LIN {X 0,Y 307.304,Z 950.743,A -85,B 0,C 180,E1 6847.604,E2 6847.604} C_VEL
LIN {X 0,Y 314.921,Z 929.321,A -85,B 0,C 180,E1 6846.872,E2 6846.872} C_VEL
LIN {X 0,Y 321.32,Z 907.161,A -85,B 0,C 180,E1 6846.28,E2 6846.28} C_VEL
LIN {X 0,Y 326.078,Z 884.655,A -85,B 0,C 180,E1 6845.831,E2 6845.831} C_VEL
LIN {X 0,Y 330.037,Z 856.626,A -85,B 0,C 180,E1 6845.371,E2 6845.371} C_VEL
LIN {X 0,Y 339.234,Z 777.222,A -85,B 0,C 180,E1 6844.099,E2 6844.099} C_VEL
LIN {X 0,Y 338.826,Z 774.8,A -85,B 0,C 180,E1 6841.353,E2 6841.353} C_VEL
LIN {X 0,Y 338.86,Z 775.076,A -85,B 0,C 180,E1 6838.648,E2 6838.648} C_VEL
LIN {X 0,Y 339.251,Z 777.523,A -85,B 0,C 180,E1 6836.249,E2 6836.249} C_VEL
LIN {X 0,Y 331.698,Z 842.7,A -85,B 0,C 180,E1 6835.221,E2 6835.221} C_VEL
LIN {X 0,Y 330.732,Z 850.398,A -85,B 0,C 180,E1 6835.274,E2 6835.274} C_VEL
LIN {X 0,Y 327.738,Z 870.97,A -85,B 0,C 180,E1 6836.04,E2 6836.04} C_VEL
LIN {X 0,Y 326.755,Z 877.56,A -85,B 0,C 180,E1 6836.062,E2 6836.062} C_VEL
LIN {X 0,Y 322.13,Z 901.741,A -85,B 0,C 180,E1 6835.656,E2 6835.656} C_VEL
LIN {X 0,Y 316.056,Z 924.847,A -85,B 0,C 180,E1 6835.216,E2 6835.216} C_VEL
LIN {X 0,Y 308.577,Z 946.561,A -85,B 0,C 180,E1 6834.679,E2 6834.679} C_VEL
LIN {X 0,Y 299.618,Z 968.19,A -85,B 0,C 180,E1 6833.966,E2 6833.966} C_VEL
LIN {X 0,Y 289.561,Z 988.431,A -85,B 0,C 180,E1 6833.093,E2 6833.093} C_VEL
LIN {X 0,Y 277.319,Z 1009.585,A -85,B 0,C 180,E1 6831.917,E2 6831.917} C_VEL
LIN {X 0,Y 265.491,Z 1027.358,A -85,B 0,C 180,E1 6830.648,E2 6830.648} C_VEL
LIN {X 0,Y 251.154,Z 1046.271,A -85,B 0,C 180,E1 6828.911,E2 6828.911} C_VEL
LIN {X 0,Y 237.094,Z 1062.776,A -85,B 0,C 180,E1 6826.946,E2 6826.946} C_VEL
LIN {X 0,Y 222.042,Z 1078.451,A -85,B 0,C 180,E1 6824.503,E2 6824.503} C_VEL
LIN {X 0,Y 206.628,Z 1093.042,A -85,B 0,C 180,E1 6821.519,E2 6821.519} C_VEL
LIN {X 0,Y 190.265,Z 1106.858,A -85,B 0,C 180,E1 6817.652,E2 6817.652} C_VEL
LIN {X 0,Y 174.199,Z 1119.33,A -85,B 0,C 180,E1 6812.83,E2 6812.83} C_VEL
LIN {X 0,Y 160.204,Z 1129.348,A -85,B 0,C 180,E1 6807.41,E2 6807.41} C_VEL
LIN {X 0,Y 145.976,Z 1139.015,A -85,B 0,C 180,E1 6799.922,E2 6799.922} C_VEL
LIN {X 0,Y 135.005,Z 1146.412,A -85,B 0,C 180,E1 6791.583,E2 6791.583} C_VEL
LIN {X 0,Y 126.79,Z 1152.12,A -85,B 0,C 180,E1 6781.894,E2 6781.894} C_VEL
LIN {X 0,Y 122.009,Z 1156.198,A -85,B 0,C 180,E1 6771.639,E2 6771.639} C_VEL
LIN {X 0,Y 120.185,Z 1158.49,A -85,B 0,C 180,E1 6761.516,E2 6761.516} C_VEL
LIN {X 0,Y 120.048,Z 1159.311,A -85,B 0,C 180,E1 6754.298,E2 6754.298} C_VEL
LIN {X 0,Y 120.076,Z 1159.432,A -85,B 0,C 180,E1 6748.09,E2 6748.09} C_VEL
LIN {X 0,Y 120.087,Z 1158.85,A -85,B 0,C 180,E1 6740.897,E2 6740.897} C_VEL
LIN {X 0,Y 121.02,Z 1157.169,A -85,B 0,C 180,E1 6732.199,E2 6732.199} C_VEL
LIN {X 0,Y 124.458,Z 1153.974,A -85,B 0,C 180,E1 6722.227,E2 6722.227} C_VEL
LIN {X 0,Y 131.118,Z 1148.973,A -85,B 0,C 180,E1 6712.405,E2 6712.405} C_VEL
LIN {X 0,Y 141.005,Z 1142.346,A -85,B 0,C 180,E1 6703.456,E2 6703.456} C_VEL
LIN {X 0,Y 153.181,Z 1134.092,A -85,B 0,C 180,E1 6695.962,E2 6695.962} C_VEL
LIN {X 0,Y 167.02,Z 1124.515,A -85,B 0,C 180,E1 6689.767,E2 6689.767} C_VEL
LIN {X 0,Y 182.454,Z 1112.942,A -85,B 0,C 180,E1 6684.535,E2 6684.535} C_VEL
LIN {X 0,Y 199.151,Z 1099.358,A -85,B 0,C 180,E1 6680.137,E2 6680.137} C_VEL
LIN {X 0,Y 214.255,Z 1085.841,A -85,B 0,C 180,E1 6676.925,E2 6676.925} C_VEL
LIN {X 0,Y 229.947,Z 1070.203,A -85,B 0,C 180,E1 6674.148,E2 6674.148} C_VEL
LIN {X 0,Y 244.761,Z 1053.844,A -85,B 0,C 180,E1 6671.935,E2 6671.935} C_VEL
LIN {X 0,Y 258.978,Z 1035.964,A -85,B 0,C 180,E1 6670.096,E2 6670.096} C_VEL
LIN {X 0,Y 272.509,Z 1016.818,A -85,B 0,C 180,E1 6668.57,E2 6668.57} C_VEL
LIN {X 0,Y 284.321,Z 997.516,A -85,B 0,C 180,E1 6667.383,E2 6667.383} C_VEL
LIN {X 0,Y 295.777,Z 975.83,A -85,B 0,C 180,E1 6666.349,E2 6666.349} C_VEL
LIN {X 0,Y 304.435,Z 956.539,A -85,B 0,C 180,E1 6665.639,E2 6665.639} C_VEL
LIN {X 0,Y 312.899,Z 933.827,A -85,B 0,C 180,E1 6664.996,E2 6664.996} C_VEL
LIN {X 0,Y 319.458,Z 911.926,A -85,B 0,C 180,E1 6664.531,E2 6664.531} C_VEL
LIN {X 0,Y 324.641,Z 888.54,A -85,B 0,C 180,E1 6664.12,E2 6664.12} C_VEL
LIN {X 0,Y 328.326,Z 864.356,A -85,B 0,C 180,E1 6663.732,E2 6663.732} C_VEL
LIN {X 0,Y 337.778,Z 783.961,A -85,B 0,C 180,E1 6662.46,E2 6662.46} C_VEL
LIN {X 0,Y 337.616,Z 782.659,A -85,B 0,C 180,E1 6660.848,E2 6660.848} C_VEL
LIN {X 0,Y 337.661,Z 782.798,A -85,B 0,C 180,E1 6658.133,E2 6658.133} C_VEL
LIN {X 0,Y 337.737,Z 784.15,A -85,B 0,C 180,E1 6657.032,E2 6657.032} C_VEL
LIN {X 0,Y 326.505,Z 877.088,A -85,B 0,C 180,E1 6655.607,E2 6655.607} C_VEL
LIN {X 0,Y 321.978,Z 900.285,A -85,B 0,C 180,E1 6655.195,E2 6655.195} C_VEL
LIN {X 0,Y 316.31,Z 921.955,A -85,B 0,C 180,E1 6654.704,E2 6654.704} C_VEL
LIN {X 0,Y 308.915,Z 943.644,A -85,B 0,C 180,E1 6654.055,E2 6654.055} C_VEL
LIN {X 0,Y 300.054,Z 965.186,A -85,B 0,C 180,E1 6653.231,E2 6653.231} C_VEL
LIN {X 0,Y 290.106,Z 985.211,A -85,B 0,C 180,E1 6652.261,E2 6652.261} C_VEL
LIN {X 0,Y 278.377,Z 1005.538,A -85,B 0,C 180,E1 6651.02,E2 6651.02} C_VEL
LIN {X 0,Y 266.782,Z 1022.943,A -85,B 0,C 180,E1 6649.681,E2 6649.681} C_VEL
LIN {X 0,Y 252.163,Z 1042.185,A -85,B 0,C 180,E1 6647.801,E2 6647.801} C_VEL
LIN {X 0,Y 238.725,Z 1057.821,A -85,B 0,C 180,E1 6645.84,E2 6645.84} C_VEL
LIN {X 0,Y 223.427,Z 1073.606,A -85,B 0,C 180,E1 6643.274,E2 6643.274} C_VEL
LIN {X 0,Y 208.212,Z 1087.758,A -85,B 0,C 180,E1 6640.26,E2 6640.26} C_VEL
LIN {X 0,Y 192.835,Z 1100.485,A -85,B 0,C 180,E1 6636.602,E2 6636.602} C_VEL
LIN {X 0,Y 177.611,Z 1112.082,A -85,B 0,C 180,E1 6632.11,E2 6632.11} C_VEL
LIN {X 0,Y 162.914,Z 1122.179,A -85,B 0,C 180,E1 6626.584,E2 6626.584} C_VEL
LIN {X 0,Y 148.74,Z 1131.321,A -85,B 0,C 180,E1 6619.431,E2 6619.431} C_VEL
LIN {X 0,Y 137.683,Z 1138.152,A -85,B 0,C 180,E1 6611.582,E2 6611.582} C_VEL
LIN {X 0,Y 128.647,Z 1143.73,A -85,B 0,C 180,E1 6601.906,E2 6601.906} C_VEL
LIN {X 0,Y 123.388,Z 1147.309,A -85,B 0,C 180,E1 6592.388,E2 6592.388} C_VEL
LIN {X 0,Y 120.712,Z 1149.56,A -85,B 0,C 180,E1 6581.952,E2 6581.952} C_VEL
LIN {X 0,Y 120.131,Z 1150.324,A -85,B 0,C 180,E1 6574.297,E2 6574.297} C_VEL
LIN {X 0,Y 120.103,Z 1150.408,A -85,B 0,C 180,E1 6567.46,E2 6567.46} C_VEL
LIN {X 0,Y 120.536,Z 1149.772,A -85,B 0,C 180,E1 6559.486,E2 6559.486} C_VEL
LIN {X 0,Y 122.361,Z 1148.099,A -85,B 0,C 180,E1 6550.427,E2 6550.427} C_VEL
LIN {X 0,Y 127.569,Z 1144.463,A -85,B 0,C 180,E1 6539.561,E2 6539.561} C_VEL
LIN {X 0,Y 135.249,Z 1139.699,A -85,B 0,C 180,E1 6530.524,E2 6530.524} C_VEL
LIN {X 0,Y 146.433,Z 1132.808,A -85,B 0,C 180,E1 6521.905,E2 6521.905} C_VEL
LIN {X 0,Y 159.565,Z 1124.556,A -85,B 0,C 180,E1 6514.829,E2 6514.829} C_VEL
LIN {X 0,Y 173.885,Z 1114.756,A -85,B 0,C 180,E1 6509.072,E2 6509.072} C_VEL
LIN {X 0,Y 189.62,Z 1103.173,A -85,B 0,C 180,E1 6504.187,E2 6504.187} C_VEL
LIN {X 0,Y 204.821,Z 1090.779,A -85,B 0,C 180,E1 6500.403,E2 6500.403} C_VEL
LIN {X 0,Y 220.887,Z 1076.247,A -85,B 0,C 180,E1 6497.112,E2 6497.112} C_VEL
LIN {X 0,Y 235.551,Z 1061.471,A -85,B 0,C 180,E1 6494.579,E2 6494.579} C_VEL
LIN {X 0,Y 250.283,Z 1044.711,A -85,B 0,C 180,E1 6492.379,E2 6492.379} C_VEL
LIN {X 0,Y 263.957,Z 1027.273,A -85,B 0,C 180,E1 6490.588,E2 6490.588} C_VEL
LIN {X 0,Y 276.451,Z 1008.884,A -85,B 0,C 180,E1 6489.113,E2 6489.113} C_VEL
LIN {X 0,Y 288.167,Z 989.301,A -85,B 0,C 180,E1 6487.861,E2 6487.861} C_VEL
LIN {X 0,Y 298.576,Z 968.744,A -85,B 0,C 180,E1 6486.83,E2 6486.83} C_VEL
LIN {X 0,Y 308.112,Z 946.386,A -85,B 0,C 180,E1 6485.944,E2 6485.944} C_VEL
LIN {X 0,Y 315.308,Z 925.792,A -85,B 0,C 180,E1 6485.31,E2 6485.31} C_VEL
LIN {X 0,Y 321.687,Z 902.515,A -85,B 0,C 180,E1 6484.757,E2 6484.757} C_VEL
LIN {X 0,Y 326.268,Z 880.083,A -85,B 0,C 180,E1 6484.348,E2 6484.348} C_VEL
LIN {X 0,Y 331.506,Z 838.837,A -85,B 0,C 180,E1 6483.708,E2 6483.708} C_VEL
LIN {X 0,Y 337.966,Z 784.117,A -85,B 0,C 180,E1 6482.841,E2 6482.841} C_VEL
LIN {X 0,Y 337.835,Z 782.731,A -85,B 0,C 180,E1 6481.187,E2 6481.187} C_VEL
LIN {X 0,Y 337.865,Z 782.963,A -85,B 0,C 180,E1 6478.813,E2 6478.813} C_VEL
LIN {X 0,Y 337.96,Z 784.492,A -85,B 0,C 180,E1 6477.496,E2 6477.496} C_VEL
LIN {X 0,Y 326.755,Z 877.56,A -85,B 0,C 180,E1 6476.062,E2 6476.062} C_VEL
LIN {X 0,Y 325.501,Z 885.224,A -85,B 0,C 180,E1 6476.117,E2 6476.117} C_VEL
LIN {X 0,Y 321.112,Z 904.429,A -85,B 0,C 180,E1 6476.864,E2 6476.864} C_VEL
LIN {X 0,Y 319.067,Z 911.917,A -85,B 0,C 180,E1 6476.908,E2 6476.908} C_VEL
LIN {X 0,Y 312.544,Z 933.468,A -85,B 0,C 180,E1 6476.483,E2 6476.483} C_VEL
LIN {X 0,Y 304.234,Z 955.616,A -85,B 0,C 180,E1 6475.904,E2 6475.904} C_VEL
LIN {X 0,Y 295.301,Z 975.326,A -85,B 0,C 180,E1 6475.233,E2 6475.233} C_VEL
LIN {X 0,Y 283.871,Z 996.758,A -85,B 0,C 180,E1 6474.284,E2 6474.284} C_VEL
LIN {X 0,Y 272.365,Z 1015.36,A -85,B 0,C 180,E1 6473.223,E2 6473.223} C_VEL
LIN {X 0,Y 258.608,Z 1034.693,A -85,B 0,C 180,E1 6471.798,E2 6471.798} C_VEL
LIN {X 0,Y 244.325,Z 1052.447,A -85,B 0,C 180,E1 6470.104,E2 6470.104} C_VEL
LIN {X 0,Y 228.972,Z 1069.145,A -85,B 0,C 180,E1 6467.999,E2 6467.999} C_VEL
LIN {X 0,Y 212.863,Z 1084.901,A -85,B 0,C 180,E1 6465.379,E2 6465.379} C_VEL
LIN {X 0,Y 197.007,Z 1098.697,A -85,B 0,C 180,E1 6462.272,E2 6462.272} C_VEL
LIN {X 0,Y 179.141,Z 1112.733,A -85,B 0,C 180,E1 6457.896,E2 6457.896} C_VEL
LIN {X 0,Y 163.015,Z 1124.291,A -85,B 0,C 180,E1 6452.792,E2 6452.792} C_VEL
LIN {X 0,Y 148.408,Z 1133.85,A -85,B 0,C 180,E1 6446.658,E2 6446.658} C_VEL
LIN {X 0,Y 135.177,Z 1142.202,A -85,B 0,C 180,E1 6438.977,E2 6438.977} C_VEL
LIN {X 0,Y 124.605,Z 1148.702,A -85,B 0,C 180,E1 6429.936,E2 6429.936} C_VEL
LIN {X 0,Y 116.939,Z 1153.86,A -85,B 0,C 180,E1 6419.166,E2 6419.166} C_VEL
LIN {X 0,Y 113.248,Z 1156.881,A -85,B 0,C 180,E1 6409.066,E2 6409.066} C_VEL
LIN {X 0,Y 112.105,Z 1158.557,A -85,B 0,C 180,E1 6399.755,E2 6399.755} C_VEL
LIN {X 0,Y 112.078,Z 1159.135,A -85,B 0,C 180,E1 6392.044,E2 6392.044} C_VEL
LIN {X 0,Y 112.049,Z 1159.006,A -85,B 0,C 180,E1 6385.392,E2 6385.392} C_VEL
LIN {X 0,Y 112.293,Z 1158.1,A -85,B 0,C 180,E1 6377.137,E2 6377.137} C_VEL
LIN {X 0,Y 114.752,Z 1155.526,A -85,B 0,C 180,E1 6365.824,E2 6365.824} C_VEL
LIN {X 0,Y 120.146,Z 1151.557,A -85,B 0,C 180,E1 6355.534,E2 6355.534} C_VEL
LIN {X 0,Y 129.836,Z 1145.41,A -85,B 0,C 180,E1 6345.11,E2 6345.11} C_VEL
LIN {X 0,Y 141.492,Z 1138.167,A -85,B 0,C 180,E1 6337.009,E2 6337.009} C_VEL
LIN {X 0,Y 156.544,Z 1128.482,A -85,B 0,C 180,E1 6329.696,E2 6329.696} C_VEL
LIN {X 0,Y 172.067,Z 1117.87,A -85,B 0,C 180,E1 6324.171,E2 6324.171} C_VEL
LIN {X 0,Y 188.065,Z 1105.777,A -85,B 0,C 180,E1 6319.771,E2 6319.771} C_VEL
LIN {X 0,Y 204.501,Z 1092.244,A -85,B 0,C 180,E1 6316.181,E2 6316.181} C_VEL
LIN {X 0,Y 219.965,Z 1077.968,A -85,B 0,C 180,E1 6313.403,E2 6313.403} C_VEL
LIN {X 0,Y 236.275,Z 1061.229,A -85,B 0,C 180,E1 6310.954,E2 6310.954} C_VEL
LIN {X 0,Y 249.797,Z 1045.606,A -85,B 0,C 180,E1 6309.213,E2 6309.213} C_VEL
LIN {X 0,Y 264.755,Z 1026.08,A -85,B 0,C 180,E1 6307.538,E2 6307.538} C_VEL
LIN {X 0,Y 276.668,Z 1008.359,A -85,B 0,C 180,E1 6306.361,E2 6306.361} C_VEL
LIN {X 0,Y 288.695,Z 987.722,A -85,B 0,C 180,E1 6305.294,E2 6305.294} C_VEL
LIN {X 0,Y 298.875,Z 967.433,A -85,B 0,C 180,E1 6304.479,E2 6304.479} C_VEL
LIN {X 0,Y 307.649,Z 946.419,A -85,B 0,C 180,E1 6303.833,E2 6303.833} C_VEL
LIN {X 0,Y 315.242,Z 924.604,A -85,B 0,C 180,E1 6303.33,E2 6303.33} C_VEL
LIN {X 0,Y 321.375,Z 901.511,A -85,B 0,C 180,E1 6302.918,E2 6302.918} C_VEL
LIN {X 0,Y 326.058,Z 877.344,A -85,B 0,C 180,E1 6302.531,E2 6302.531} C_VEL
LIN {X 0,Y 336.668,Z 790.79,A -85,B 0,C 180,E1 6301.222,E2 6301.222} C_VEL
LIN {X 0,Y 336.65,Z 790.83,A -85,B 0,C 180,E1 6298.295,E2 6298.295} C_VEL
LIN {X 0,Y 325.954,Z 877.666,A -85,B 0,C 180,E1 6297.005,E2 6297.005} C_VEL
LIN {X 0,Y 321.376,Z 900.726,A -85,B 0,C 180,E1 6296.615,E2 6296.615} C_VEL
LIN {X 0,Y 315.428,Z 923.072,A -85,B 0,C 180,E1 6296.132,E2 6296.132} C_VEL
LIN {X 0,Y 307.903,Z 944.7,A -85,B 0,C 180,E1 6295.516,E2 6295.516} C_VEL
LIN {X 0,Y 298.729,Z 966.492,A -85,B 0,C 180,E1 6294.72,E2 6294.72} C_VEL
LIN {X 0,Y 289.139,Z 985.504,A -85,B 0,C 180,E1 6293.846,E2 6293.846} C_VEL
LIN {X 0,Y 277.23,Z 1005.846,A -85,B 0,C 180,E1 6292.672,E2 6292.672} C_VEL
LIN {X 0,Y 265.592,Z 1023.048,A -85,B 0,C 180,E1 6291.423,E2 6291.423} C_VEL
LIN {X 0,Y 250.946,Z 1042.045,A -85,B 0,C 180,E1 6289.671,E2 6289.671} C_VEL
LIN {X 0,Y 237.31,Z 1057.631,A -85,B 0,C 180,E1 6287.824,E2 6287.824} C_VEL
LIN {X 0,Y 221.205,Z 1073.917,A -85,B 0,C 180,E1 6285.309,E2 6285.309} C_VEL
LIN {X 0,Y 205.579,Z 1088.069,A -85,B 0,C 180,E1 6282.418,E2 6282.418} C_VEL
LIN {X 0,Y 189.711,Z 1100.796,A -85,B 0,C 180,E1 6278.889,E2 6278.889} C_VEL
LIN {X 0,Y 173.459,Z 1112.68,A -85,B 0,C 180,E1 6274.385,E2 6274.385} C_VEL
LIN {X 0,Y 158.507,Z 1122.491,A -85,B 0,C 180,E1 6269.082,E2 6269.082} C_VEL
LIN {X 0,Y 143.497,Z 1131.632,A -85,B 0,C 180,E1 6261.941,E2 6261.941} C_VEL
LIN {X 0,Y 131.914,Z 1138.284,A -85,B 0,C 180,E1 6254.214,E2 6254.214} C_VEL
LIN {X 0,Y 121.749,Z 1144.039,A -85,B 0,C 180,E1 6243.95,E2 6243.95} C_VEL
LIN {X 0,Y 115.679,Z 1147.767,A -85,B 0,C 180,E1 6233.429,E2 6233.429} C_VEL
LIN {X 0,Y 112.813,Z 1149.864,A -85,B 0,C 180,E1 6222.803,E2 6222.803} C_VEL
LIN {X 0,Y 112.147,Z 1150.624,A -85,B 0,C 180,E1 6214.604,E2 6214.604} C_VEL
LIN {X 0,Y 112.108,Z 1150.709,A -85,B 0,C 180,E1 6207.322,E2 6207.322} C_VEL
LIN {X 0,Y 112.559,Z 1150.137,A -85,B 0,C 180,E1 6199.25,E2 6199.25} C_VEL
LIN {X 0,Y 114.395,Z 1148.616,A -85,B 0,C 180,E1 6190.071,E2 6190.071} C_VEL
LIN {X 0,Y 119.724,Z 1145.292,A -85,B 0,C 180,E1 6178.817,E2 6178.817} C_VEL
LIN {X 0,Y 127.629,Z 1140.739,A -85,B 0,C 180,E1 6169.442,E2 6169.442} C_VEL
LIN {X 0,Y 139.883,Z 1133.801,A -85,B 0,C 180,E1 6160.11,E2 6160.11} C_VEL
LIN {X 0,Y 152.96,Z 1126.055,A -85,B 0,C 180,E1 6153.207,E2 6153.207} C_VEL
LIN {X 0,Y 168.523,Z 1116.07,A -85,B 0,C 180,E1 6147.132,E2 6147.132} C_VEL
LIN {X 0,Y 183.984,Z 1105.302,A -85,B 0,C 180,E1 6142.503,E2 6142.503} C_VEL
LIN {X 0,Y 199.983,Z 1092.808,A -85,B 0,C 180,E1 6138.662,E2 6138.662} C_VEL
LIN {X 0,Y 215.864,Z 1079.167,A -85,B 0,C 180,E1 6135.543,E2 6135.543} C_VEL
LIN {X 0,Y 231.216,Z 1064.217,A -85,B 0,C 180,E1 6132.996,E2 6132.996} C_VEL
LIN {X 0,Y 246.823,Z 1047.208,A -85,B 0,C 180,E1 6130.783,E2 6130.783} C_VEL
LIN {X 0,Y 260.246,Z 1030.584,A -85,B 0,C 180,E1 6129.111,E2 6129.111} C_VEL
LIN {X 0,Y 273.865,Z 1011.368,A -85,B 0,C 180,E1 6127.596,E2 6127.596} C_VEL
LIN {X 0,Y 285.349,Z 992.767,A -85,B 0,C 180,E1 6126.438,E2 6126.438} C_VEL
LIN {X 0,Y 296.282,Z 972.035,A -85,B 0,C 180,E1 6125.42,E2 6125.42} C_VEL
LIN {X 0,Y 305.451,Z 951.658,A -85,B 0,C 180,E1 6124.625,E2 6124.625} C_VEL
LIN {X 0,Y 313.355,Z 930.06,A -85,B 0,C 180,E1 6123.963,E2 6123.963} C_VEL
LIN {X 0,Y 319.874,Z 908.122,A -85,B 0,C 180,E1 6123.436,E2 6123.436} C_VEL
LIN {X 0,Y 324.812,Z 885.385,A -85,B 0,C 180,E1 6123.024,E2 6123.024} C_VEL
LIN {X 0,Y 328.839,Z 857.901,A -85,B 0,C 180,E1 6122.604,E2 6122.604} C_VEL
LIN {X 0,Y 336.875,Z 790.916,A -85,B 0,C 180,E1 6121.574,E2 6121.574} C_VEL
LIN {X 0,Y 336.873,Z 790.849,A -85,B 0,C 180,E1 6118.98,E2 6118.98} C_VEL
LIN {X 0,Y 336.844,Z 791.345,A -85,B 0,C 180,E1 6118.754,E2 6118.754} C_VEL
LIN {X 0,Y 326.089,Z 878.773,A -85,B 0,C 180,E1 6117.45,E2 6117.45} C_VEL
LIN {X 0,Y 321.406,Z 902.367,A -85,B 0,C 180,E1 6117.071,E2 6117.071} C_VEL
LIN {X 0,Y 319.067,Z 911.917,A -85,B 0,C 180,E1 6116.908,E2 6116.908} C_VEL
LIN {X 0,Y 316.904,Z 919.36,A -85,B 0,C 180,E1 6116.972,E2 6116.972} C_VEL
LIN {X 0,Y 310.573,Z 938.034,A -85,B 0,C 180,E1 6117.714,E2 6117.714} C_VEL
LIN {X 0,Y 307.761,Z 945.289,A -85,B 0,C 180,E1 6117.695,E2 6117.695} C_VEL
LIN {X 0,Y 298.842,Z 966.585,A -85,B 0,C 180,E1 6117.094,E2 6117.094} C_VEL
LIN {X 0,Y 288.244,Z 987.488,A -85,B 0,C 180,E1 6116.319,E2 6116.319} C_VEL
LIN {X 0,Y 275.883,Z 1008.394,A -85,B 0,C 180,E1 6115.314,E2 6115.314} C_VEL
LIN {X 0,Y 263.804,Z 1026.077,A -85,B 0,C 180,E1 6114.218,E2 6114.218} C_VEL
LIN {X 0,Y 248.986,Z 1045.099,A -85,B 0,C 180,E1 6112.694,E2 6112.694} C_VEL
LIN {X 0,Y 234.845,Z 1061.136,A -85,B 0,C 180,E1 6111.02,E2 6111.02} C_VEL
LIN {X 0,Y 219.105,Z 1076.976,A -85,B 0,C 180,E1 6108.849,E2 6108.849} C_VEL
LIN {X 0,Y 203.74,Z 1090.856,A -85,B 0,C 180,E1 6106.332,E2 6106.332} C_VEL
LIN {X 0,Y 186.261,Z 1104.94,A -85,B 0,C 180,E1 6102.845,E2 6102.845} C_VEL
LIN {X 0,Y 169.034,Z 1117.502,A -85,B 0,C 180,E1 6098.486,E2 6098.486} C_VEL
LIN {X 0,Y 152.563,Z 1128.251,A -85,B 0,C 180,E1 6093.037,E2 6093.037} C_VEL
LIN {X 0,Y 136.211,Z 1138.143,A -85,B 0,C 180,E1 6085.584,E2 6085.584} C_VEL
LIN {X 0,Y 123.71,Z 1145.352,A -85,B 0,C 180,E1 6077.347,E2 6077.347} C_VEL
LIN {X 0,Y 113.387,Z 1151.28,A -85,B 0,C 180,E1 6066.842,E2 6066.842} C_VEL
LIN {X 0,Y 107.073,Z 1155.414,A -85,B 0,C 180,E1 6055.438,E2 6055.438} C_VEL
LIN {X 0,Y 104.383,Z 1157.807,A -85,B 0,C 180,E1 6043.854,E2 6043.854} C_VEL
LIN {X 0,Y 104.046,Z 1158.683,A -85,B 0,C 180,E1 6035.513,E2 6035.513} C_VEL
LIN {X 0,Y 104.088,Z 1158.856,A -85,B 0,C 180,E1 6028.347,E2 6028.347} C_VEL
LIN {X 0,Y 104.112,Z 1158.316,A -85,B 0,C 180,E1 6020.044,E2 6020.044} C_VEL
LIN {X 0,Y 105.448,Z 1156.632,A -85,B 0,C 180,E1 6009.833,E2 6009.833} C_VEL
LIN {X 0,Y 109.782,Z 1153.522,A -85,B 0,C 180,E1 5998.724,E2 5998.724} C_VEL
LIN {X 0,Y 118.321,Z 1148.345,A -85,B 0,C 180,E1 5987.464,E2 5987.464} C_VEL
LIN {X 0,Y 129.828,Z 1141.832,A -85,B 0,C 180,E1 5978.227,E2 5978.227} C_VEL
LIN {X 0,Y 144.319,Z 1133.244,A -85,B 0,C 180,E1 5970.38,E2 5970.38} C_VEL
LIN {X 0,Y 160.125,Z 1123.355,A -85,B 0,C 180,E1 5964.262,E2 5964.262} C_VEL
LIN {X 0,Y 176.208,Z 1112.275,A -85,B 0,C 180,E1 5959.559,E2 5959.559} C_VEL
LIN {X 0,Y 194.03,Z 1098.727,A -85,B 0,C 180,E1 5955.496,E2 5955.496} C_VEL
LIN {X 0,Y 210.01,Z 1085.211,A -85,B 0,C 180,E1 5952.573,E2 5952.573} C_VEL
LIN {X 0,Y 226.466,Z 1069.576,A -85,B 0,C 180,E1 5950.078,E2 5950.078} C_VEL
LIN {X 0,Y 242.218,Z 1052.856,A -85,B 0,C 180,E1 5948.067,E2 5948.067} C_VEL
LIN {X 0,Y 256.607,Z 1035.34,A -85,B 0,C 180,E1 5946.48,E2 5946.48} C_VEL
LIN {X 0,Y 270.554,Z 1016.195,A -85,B 0,C 180,E1 5945.14,E2 5945.14} C_VEL
LIN {X 0,Y 282.689,Z 996.894,A -85,B 0,C 180,E1 5944.103,E2 5944.103} C_VEL
LIN {X 0,Y 294.423,Z 975.209,A -85,B 0,C 180,E1 5943.206,E2 5943.206} C_VEL
LIN {X 0,Y 303.272,Z 955.918,A -85,B 0,C 180,E1 5942.595,E2 5942.595} C_VEL
LIN {X 0,Y 311.909,Z 933.204,A -85,B 0,C 180,E1 5942.044,E2 5942.044} C_VEL
LIN {X 0,Y 318.529,Z 911.517,A -85,B 0,C 180,E1 5941.647,E2 5941.647} C_VEL
LIN {X 0,Y 323.852,Z 888.067,A -85,B 0,C 180,E1 5941.281,E2 5941.281} C_VEL
LIN {X 0,Y 327.641,Z 863.956,A -85,B 0,C 180,E1 5940.925,E2 5940.925} C_VEL
LIN {X 0,Y 335.605,Z 798.522,A -85,B 0,C 180,E1 5939.957,E2 5939.957} C_VEL
LIN {X 0,Y 335.581,Z 798.71,A -85,B 0,C 180,E1 5939.549,E2 5939.549} C_VEL
LIN {X 0,Y 325.6,Z 878.223,A -85,B 0,C 180,E1 5938.407,E2 5938.407} C_VEL
LIN {X 0,Y 320.973,Z 901.168,A -85,B 0,C 180,E1 5938.039,E2 5938.039} C_VEL
LIN {X 0,Y 314.989,Z 923.383,A -85,B 0,C 180,E1 5937.588,E2 5937.588} C_VEL
LIN {X 0,Y 307.38,Z 945.01,A -85,B 0,C 180,E1 5937.008,E2 5937.008} C_VEL
LIN {X 0,Y 298.097,Z 966.801,A -85,B 0,C 180,E1 5936.261,E2 5936.261} C_VEL
LIN {X 0,Y 288.199,Z 986.156,A -85,B 0,C 180,E1 5935.423,E2 5935.423} C_VEL
LIN {X 0,Y 275.833,Z 1006.882,A -85,B 0,C 180,E1 5934.291,E2 5934.291} C_VEL
LIN {X 0,Y 263.88,Z 1024.221,A -85,B 0,C 180,E1 5933.096,E2 5933.096} C_VEL
LIN {X 0,Y 249.195,Z 1042.842,A -85,B 0,C 180,E1 5931.462,E2 5931.462} C_VEL
LIN {X 0,Y 235.399,Z 1058.289,A -85,B 0,C 180,E1 5929.723,E2 5929.723} C_VEL
LIN {X 0,Y 219.269,Z 1074.227,A -85,B 0,C 180,E1 5927.383,E2 5927.383} C_VEL
LIN {X 0,Y 202.936,Z 1088.649,A -85,B 0,C 180,E1 5924.57,E2 5924.57} C_VEL
LIN {X 0,Y 186.057,Z 1101.73,A -85,B 0,C 180,E1 5921.055,E2 5921.055} C_VEL
LIN {X 0,Y 168.913,Z 1113.711,A -85,B 0,C 180,E1 5916.566,E2 5916.566} C_VEL
LIN {X 0,Y 153.688,Z 1123.25,A -85,B 0,C 180,E1 5911.438,E2 5911.438} C_VEL
LIN {X 0,Y 137.907,Z 1132.286,A -85,B 0,C 180,E1 5904.296,E2 5904.296} C_VEL
LIN {X 0,Y 125.067,Z 1139.18,A -85,B 0,C 180,E1 5896.016,E2 5896.016} C_VEL
LIN {X 0,Y 114.637,Z 1144.545,A -85,B 0,C 180,E1 5885.76,E2 5885.76} C_VEL
LIN {X 0,Y 108.013,Z 1148.225,A -85,B 0,C 180,E1 5874.619,E2 5874.619} C_VEL
LIN {X 0,Y 104.861,Z 1150.229,A -85,B 0,C 180,E1 5863.23,E2 5863.23} C_VEL
LIN {X 0,Y 104.144,Z 1150.945,A -85,B 0,C 180,E1 5854.406,E2 5854.406} C_VEL
LIN {X 0,Y 104.115,Z 1151.011,A -85,B 0,C 180,E1 5847.159,E2 5847.159} C_VEL
LIN {X 0,Y 104.645,Z 1150.439,A -85,B 0,C 180,E1 5838.426,E2 5838.426} C_VEL
LIN {X 0,Y 106.777,Z 1148.921,A -85,B 0,C 180,E1 5828.581,E2 5828.581} C_VEL
LIN {X 0,Y 112.78,Z 1145.599,A -85,B 0,C 180,E1 5816.657,E2 5816.657} C_VEL
LIN {X 0,Y 121.478,Z 1141.048,A -85,B 0,C 180,E1 5806.911,E2 5806.911} C_VEL
LIN {X 0,Y 134.699,Z 1134.11,A -85,B 0,C 180,E1 5797.416,E2 5797.416} C_VEL
LIN {X 0,Y 148.587,Z 1126.364,A -85,B 0,C 180,E1 5790.535,E2 5790.535} C_VEL
LIN {X 0,Y 164.915,Z 1116.379,A -85,B 0,C 180,E1 5784.574,E2 5784.574} C_VEL
LIN {X 0,Y 181.397,Z 1105.327,A -85,B 0,C 180,E1 5779.984,E2 5779.984} C_VEL
LIN {X 0,Y 197.938,Z 1092.768,A -85,B 0,C 180,E1 5776.31,E2 5776.31} C_VEL
LIN {X 0,Y 214.705,Z 1078.639,A -85,B 0,C 180,E1 5773.273,E2 5773.273} C_VEL
LIN {X 0,Y 230.133,Z 1063.906,A -85,B 0,C 180,E1 5770.918,E2 5770.918} C_VEL
LIN {X 0,Y 246.364,Z 1046.413,A -85,B 0,C 180,E1 5768.799,E2 5768.799} C_VEL
LIN {X 0,Y 260.033,Z 1029.681,A -85,B 0,C 180,E1 5767.234,E2 5767.234} C_VEL
LIN {X 0,Y 273.391,Z 1010.938,A -85,B 0,C 180,E1 5765.864,E2 5765.864} C_VEL
LIN {X 0,Y 285.277,Z 991.866,A -85,B 0,C 180,E1 5764.759,E2 5764.759} C_VEL
LIN {X 0,Y 295.973,Z 971.628,A -85,B 0,C 180,E1 5763.836,E2 5763.836} C_VEL
LIN {X 0,Y 305.398,Z 950.797,A -85,B 0,C 180,E1 5763.08,E2 5763.08} C_VEL
LIN {X 0,Y 313.247,Z 929.321,A -85,B 0,C 180,E1 5762.471,E2 5762.471} C_VEL
LIN {X 0,Y 319.819,Z 907.043,A -85,B 0,C 180,E1 5761.977,E2 5761.977} C_VEL
LIN {X 0,Y 324.609,Z 885.036,A -85,B 0,C 180,E1 5761.603,E2 5761.603} C_VEL
LIN {X 0,Y 329.038,Z 854.344,A -85,B 0,C 180,E1 5761.155,E2 5761.155} C_VEL
LIN {X 0,Y 335.84,Z 798.602,A -85,B 0,C 180,E1 5760.342,E2 5760.342} C_VEL
LIN {X 0,Y 335.817,Z 798.811,A -85,B 0,C 180,E1 5760.012,E2 5760.012} C_VEL
LIN {X 0,Y 325.8,Z 878.707,A -85,B 0,C 180,E1 5758.86,E2 5758.86} C_VEL
LIN {X 0,Y 321.064,Z 902.209,A -85,B 0,C 180,E1 5758.503,E2 5758.503} C_VEL
LIN {X 0,Y 314.874,Z 925.007,A -85,B 0,C 180,E1 5758.123,E2 5758.123} C_VEL
LIN {X 0,Y 307.761,Z 945.289,A -85,B 0,C 180,E1 5757.695,E2 5757.695} C_VEL
LIN {X 0,Y 304.859,Z 952.654,A -85,B 0,C 180,E1 5757.699,E2 5757.699} C_VEL
LIN {X 0,Y 296.472,Z 970.607,A -85,B 0,C 180,E1 5758.327,E2 5758.327} C_VEL
LIN {X 0,Y 293.07,Z 977.439,A -85,B 0,C 180,E1 5758.292,E2 5758.292} C_VEL
LIN {X 0,Y 281.728,Z 997.792,A -85,B 0,C 180,E1 5757.499,E2 5757.499} C_VEL
LIN {X 0,Y 269.454,Z 1016.979,A -85,B 0,C 180,E1 5756.537,E2 5756.537} C_VEL
LIN {X 0,Y 255.81,Z 1035.313,A -85,B 0,C 180,E1 5755.337,E2 5755.337} C_VEL
LIN {X 0,Y 241.342,Z 1052.622,A -85,B 0,C 180,E1 5753.878,E2 5753.878} C_VEL
LIN {X 0,Y 226.109,Z 1068.53,A -85,B 0,C 180,E1 5752.107,E2 5752.107} C_VEL
LIN {X 0,Y 209.284,Z 1084.282,A -85,B 0,C 180,E1 5749.79,E2 5749.79} C_VEL
LIN {X 0,Y 192.867,Z 1097.846,A -85,B 0,C 180,E1 5747.064,E2 5747.064} C_VEL
LIN {X 0,Y 174.389,Z 1111.522,A -85,B 0,C 180,E1 5743.233,E2 5743.233} C_VEL
LIN {X 0,Y 157.674,Z 1122.61,A -85,B 0,C 180,E1 5738.774,E2 5738.774} C_VEL
LIN {X 0,Y 140.612,Z 1132.805,A -85,B 0,C 180,E1 5732.727,E2 5732.727} C_VEL
LIN {X 0,Y 125.45,Z 1141.252,A -85,B 0,C 180,E1 5725.177,E2 5725.177} C_VEL
LIN {X 0,Y 112.812,Z 1147.812,A -85,B 0,C 180,E1 5715.881,E2 5715.881} C_VEL
LIN {X 0,Y 103.105,Z 1153.069,A -85,B 0,C 180,E1 5704.225,E2 5704.225} C_VEL
LIN {X 0,Y 97.893,Z 1156.266,A -85,B 0,C 180,E1 5692.203,E2 5692.203} C_VEL
LIN {X 0,Y 96.143,Z 1158.024,A -85,B 0,C 180,E1 5680.788,E2 5680.788} C_VEL
LIN {X 0,Y 96.09,Z 1158.56,A -85,B 0,C 180,E1 5671.788,E2 5671.788} C_VEL
LIN {X 0,Y 96.051,Z 1158.378,A -85,B 0,C 180,E1 5664.024,E2 5664.024} C_VEL
LIN {X 0,Y 96.652,Z 1157.338,A -85,B 0,C 180,E1 5653.779,E2 5653.779} C_VEL
LIN {X 0,Y 100.431,Z 1154.568,A -85,B 0,C 180,E1 5640.8,E2 5640.8} C_VEL
LIN {X 0,Y 107.683,Z 1150.497,A -85,B 0,C 180,E1 5629.459,E2 5629.459} C_VEL
LIN {X 0,Y 119.932,Z 1144.037,A -85,B 0,C 180,E1 5618.4,E2 5618.4} C_VEL
LIN {X 0,Y 134.151,Z 1136.439,A -85,B 0,C 180,E1 5610.164,E2 5610.164} C_VEL
LIN {X 0,Y 150.498,Z 1126.906,A -85,B 0,C 180,E1 5603.531,E2 5603.531} C_VEL
LIN {X 0,Y 167.629,Z 1116.066,A -85,B 0,C 180,E1 5598.428,E2 5598.428} C_VEL
LIN {X 0,Y 183.968,Z 1104.498,A -85,B 0,C 180,E1 5594.661,E2 5594.661} C_VEL
LIN {X 0,Y 201.931,Z 1090.379,A -85,B 0,C 180,E1 5591.36,E2 5591.36} C_VEL
LIN {X 0,Y 217.755,Z 1076.385,A -85,B 0,C 180,E1 5588.981,E2 5588.981} C_VEL
LIN {X 0,Y 235.123,Z 1059.063,A -85,B 0,C 180,E1 5586.799,E2 5586.799} C_VEL
LIN {X 0,Y 250.004,Z 1042.293,A -85,B 0,C 180,E1 5585.215,E2 5585.215} C_VEL
LIN {X 0,Y 264.08,Z 1024.109,A -85,B 0,C 180,E1 5583.907,E2 5583.907} C_VEL
LIN {X 0,Y 276.763,Z 1005.59,A -85,B 0,C 180,E1 5582.874,E2 5582.874} C_VEL
LIN {X 0,Y 288.145,Z 986.195,A -85,B 0,C 180,E1 5582.034,E2 5582.034} C_VEL
LIN {X 0,Y 298.56,Z 965.765,A -85,B 0,C 180,E1 5581.343,E2 5581.343} C_VEL
LIN {X 0,Y 307.49,Z 944.507,A -85,B 0,C 180,E1 5580.794,E2 5580.794} C_VEL
LIN {X 0,Y 315.347,Z 921.844,A -85,B 0,C 180,E1 5580.363,E2 5580.363} C_VEL
LIN {X 0,Y 321.268,Z 899.587,A -85,B 0,C 180,E1 5580.027,E2 5580.027} C_VEL
LIN {X 0,Y 324.868,Z 882.043,A -85,B 0,C 180,E1 5579.765,E2 5579.765} C_VEL
LIN {X 0,Y 320.225,Z 903.872,A -85,B 0,C 180,E1 5579.427,E2 5579.427} C_VEL
LIN {X 0,Y 313.512,Z 927.377,A -85,B 0,C 180,E1 5578.959,E2 5578.959} C_VEL
LIN {X 0,Y 306.076,Z 947.874,A -85,B 0,C 180,E1 5578.431,E2 5578.431} C_VEL
LIN {X 0,Y 296.201,Z 970.104,A -85,B 0,C 180,E1 5577.697,E2 5577.697} C_VEL
LIN {X 0,Y 285.398,Z 990.603,A -85,B 0,C 180,E1 5576.839,E2 5576.839} C_VEL
LIN {X 0,Y 273.244,Z 1010.037,A -85,B 0,C 180,E1 5575.803,E2 5575.803} C_VEL
LIN {X 0,Y 260.136,Z 1028.438,A -85,B 0,C 180,E1 5574.566,E2 5574.566} C_VEL
LIN {X 0,Y 246.113,Z 1045.458,A -85,B 0,C 180,E1 5573.102,E2 5573.102} C_VEL
LIN {X 0,Y 230.65,Z 1062.12,A -85,B 0,C 180,E1 5571.259,E2 5571.259} C_VEL
LIN {X 0,Y 214.862,Z 1077.035,A -85,B 0,C 180,E1 5569.083,E2 5569.083} C_VEL
LIN {X 0,Y 196.739,Z 1092.181,A -85,B 0,C 180,E1 5566.098,E2 5566.098} C_VEL
LIN {X 0,Y 180.095,Z 1104.533,A -85,B 0,C 180,E1 5562.733,E2 5562.733} C_VEL
LIN {X 0,Y 162.995,Z 1115.746,A -85,B 0,C 180,E1 5558.403,E2 5558.403} C_VEL
LIN {X 0,Y 146.875,Z 1125.348,A -85,B 0,C 180,E1 5553.101,E2 5553.101} C_VEL
LIN {X 0,Y 131.231,Z 1133.623,A -85,B 0,C 180,E1 5546.151,E2 5546.151} C_VEL
LIN {X 0,Y 117.257,Z 1140.544,A -85,B 0,C 180,E1 5537.168,E2 5537.168} C_VEL
LIN {X 0,Y 107.246,Z 1145.248,A -85,B 0,C 180,E1 5527.303,E2 5527.303} C_VEL
LIN {X 0,Y 99.692,Z 1148.977,A -85,B 0,C 180,E1 5514.282,E2 5514.282} C_VEL
LIN {X 0,Y 96.833,Z 1150.657,A -85,B 0,C 180,E1 5503.132,E2 5503.132} C_VEL
LIN {X 0,Y 96.128,Z 1151.286,A -85,B 0,C 180,E1 5493.579,E2 5493.579} C_VEL
LIN {X 0,Y 96.139,Z 1151.273,A -85,B 0,C 180,E1 5485.826,E2 5485.826} C_VEL
LIN {X 0,Y 96.903,Z 1150.617,A -85,B 0,C 180,E1 5476.273,E2 5476.273} C_VEL
LIN {X 0,Y 100.121,Z 1148.803,A -85,B 0,C 180,E1 5464.57,E2 5464.57} C_VEL
LIN {X 0,Y 107.6,Z 1145.118,A -85,B 0,C 180,E1 5452.173,E2 5452.173} C_VEL
LIN {X 0,Y 118.847,Z 1139.878,A -85,B 0,C 180,E1 5441.518,E2 5441.518} C_VEL
LIN {X 0,Y 132.494,Z 1133.052,A -85,B 0,C 180,E1 5433.108,E2 5433.108} C_VEL
LIN {X 0,Y 148.309,Z 1124.595,A -85,B 0,C 180,E1 5426.28,E2 5426.28} C_VEL
LIN {X 0,Y 164.087,Z 1115.179,A -85,B 0,C 180,E1 5421.205,E2 5421.205} C_VEL
LIN {X 0,Y 182.612,Z 1102.85,A -85,B 0,C 180,E1 5416.63,E2 5416.63} C_VEL
LIN {X 0,Y 199.531,Z 1090.194,A -85,B 0,C 180,E1 5413.328,E2 5413.328} C_VEL
LIN {X 0,Y 215.974,Z 1076.222,A -85,B 0,C 180,E1 5410.672,E2 5410.672} C_VEL
LIN {X 0,Y 231.54,Z 1061.469,A -85,B 0,C 180,E1 5408.55,E2 5408.55} C_VEL
LIN {X 0,Y 246.761,Z 1044.973,A -85,B 0,C 180,E1 5406.749,E2 5406.749} C_VEL
LIN {X 0,Y 261.065,Z 1027.545,A -85,B 0,C 180,E1 5405.266,E2 5405.266} C_VEL
LIN {X 0,Y 274.143,Z 1009.052,A -85,B 0,C 180,E1 5404.042,E2 5404.042} C_VEL
LIN {X 0,Y 286.4,Z 989.212,A -85,B 0,C 180,E1 5403.002,E2 5403.002} C_VEL
LIN {X 0,Y 296.675,Z 969.632,A -85,B 0,C 180,E1 5402.191,E2 5402.191} C_VEL
LIN {X 0,Y 306.76,Z 946.737,A -85,B 0,C 180,E1 5401.442,E2 5401.442} C_VEL
LIN {X 0,Y 314.286,Z 925.809,A -85,B 0,C 180,E1 5400.912,E2 5400.912} C_VEL
LIN {X 0,Y 320.715,Z 902.857,A -85,B 0,C 180,E1 5400.465,E2 5400.465} C_VEL
LIN {X 0,Y 324.507,Z 885.204,A -85,B 0,C 180,E1 5400.18,E2 5400.18} C_VEL
LIN {X 0,Y 319.474,Z 908.115,A -85,B 0,C 180,E1 5399.848,E2 5399.848} C_VEL
LIN {X 0,Y 312.693,Z 930.728,A -85,B 0,C 180,E1 5399.479,E2 5399.479} C_VEL
LIN {X 0,Y 304.502,Z 952.752,A -85,B 0,C 180,E1 5399.013,E2 5399.013} C_VEL
LIN {X 0,Y 295.069,Z 973.359,A -85,B 0,C 180,E1 5398.429,E2 5398.429} C_VEL
LIN {X 0,Y 293.07,Z 977.439,A -85,B 0,C 180,E1 5398.292,E2 5398.292} C_VEL
LIN {X 0,Y 289.494,Z 984.33,A -85,B 0,C 180,E1 5398.243,E2 5398.243} C_VEL
LIN {X 0,Y 279.225,Z 1001.427,A -85,B 0,C 180,E1 5398.783,E2 5398.783} C_VEL
LIN {X 0,Y 274.968,Z 1007.885,A -85,B 0,C 180,E1 5398.701,E2 5398.701} C_VEL
LIN {X 0,Y 262.66,Z 1025.471,A -85,B 0,C 180,E1 5397.78,E2 5397.78} C_VEL
LIN {X 0,Y 247.431,Z 1044.488,A -85,B 0,C 180,E1 5396.481,E2 5396.481} C_VEL
LIN {X 0,Y 232.353,Z 1061.035,A -85,B 0,C 180,E1 5394.993,E2 5394.993} C_VEL
LIN {X 0,Y 215.555,Z 1077.216,A -85,B 0,C 180,E1 5393.046,E2 5393.046} C_VEL
LIN {X 0,Y 198.592,Z 1091.802,A -85,B 0,C 180,E1 5390.682,E2 5390.682} C_VEL
LIN {X 0,Y 181.126,Z 1104.964,A -85,B 0,C 180,E1 5387.708,E2 5387.708} C_VEL
LIN {X 0,Y 163.388,Z 1117.024,A -85,B 0,C 180,E1 5383.896,E2 5383.896} C_VEL
LIN {X 0,Y 145.716,Z 1127.624,A -85,B 0,C 180,E1 5378.936,E2 5378.936} C_VEL
LIN {X 0,Y 127.926,Z 1137.291,A -85,B 0,C 180,E1 5372.029,E2 5372.029} C_VEL
LIN {X 0,Y 113.656,Z 1144.411,A -85,B 0,C 180,E1 5364.031,E2 5364.031} C_VEL
LIN {X 0,Y 100.715,Z 1150.582,A -85,B 0,C 180,E1 5352.725,E2 5352.725} C_VEL
LIN {X 0,Y 92.434,Z 1154.796,A -85,B 0,C 180,E1 5339.839,E2 5339.839} C_VEL
LIN {X 0,Y 88.562,Z 1157.272,A -85,B 0,C 180,E1 5325.72,E2 5325.72} C_VEL
LIN {X 0,Y 88.055,Z 1158.107,A -85,B 0,C 180,E1 5315.864,E2 5315.864} C_VEL
LIN {X 0,Y 88.091,Z 1158.255,A -85,B 0,C 180,E1 5308.047,E2 5308.047} C_VEL
LIN {X 0,Y 88.156,Z 1157.782,A -85,B 0,C 180,E1 5298.881,E2 5298.881} C_VEL
LIN {X 0,Y 90.151,Z 1156.06,A -85,B 0,C 180,E1 5286.466,E2 5286.466} C_VEL
LIN {X 0,Y 95.974,Z 1152.898,A -85,B 0,C 180,E1 5273.569,E2 5273.569} C_VEL
LIN {X 0,Y 106.611,Z 1147.717,A -85,B 0,C 180,E1 5261.383,E2 5261.383} C_VEL
LIN {X 0,Y 120.855,Z 1140.871,A -85,B 0,C 180,E1 5251.552,E2 5251.552} C_VEL
LIN {X 0,Y 137.037,Z 1132.371,A -85,B 0,C 180,E1 5244.115,E2 5244.115} C_VEL
LIN {X 0,Y 154.833,Z 1122.195,A -85,B 0,C 180,E1 5238.324,E2 5238.324} C_VEL
LIN {X 0,Y 172.159,Z 1111.092,A -85,B 0,C 180,E1 5234.09,E2 5234.09} C_VEL
LIN {X 0,Y 191.172,Z 1097.383,A -85,B 0,C 180,E1 5230.491,E2 5230.491} C_VEL
LIN {X 0,Y 208.918,Z 1083.014,A -85,B 0,C 180,E1 5227.821,E2 5227.821} C_VEL
LIN {X 0,Y 225.123,Z 1068.011,A -85,B 0,C 180,E1 5225.797,E2 5225.797} C_VEL
LIN {X 0,Y 241.091,Z 1051.523,A -85,B 0,C 180,E1 5224.113,E2 5224.113} C_VEL
LIN {X 0,Y 255.562,Z 1034.359,A -85,B 0,C 180,E1 5222.791,E2 5222.791} C_VEL
LIN {X 0,Y 270.076,Z 1014.832,A -85,B 0,C 180,E1 5221.64,E2 5221.64} C_VEL
LIN {X 0,Y 281.992,Z 996.273,A -85,B 0,C 180,E1 5220.799,E2 5220.799} C_VEL
LIN {X 0,Y 293.963,Z 974.587,A -85,B 0,C 180,E1 5220.045,E2 5220.045} C_VEL
LIN {X 0,Y 301.34,Z 958.996,A -85,B 0,C 180,E1 5219.619,E2 5219.619} C_VEL
LIN {X 0,Y 291.017,Z 980.191,A -85,B 0,C 180,E1 5218.895,E2 5218.895} C_VEL
LIN {X 0,Y 280.12,Z 999.01,A -85,B 0,C 180,E1 5218.087,E2 5218.087} C_VEL
LIN {X 0,Y 266.34,Z 1019.549,A -85,B 0,C 180,E1 5216.963,E2 5216.963} C_VEL
LIN {X 0,Y 253.157,Z 1036.573,A -85,B 0,C 180,E1 5215.772,E2 5215.772} C_VEL
LIN {X 0,Y 237.206,Z 1054.557,A -85,B 0,C 180,E1 5214.149,E2 5214.149} C_VEL
LIN {X 0,Y 220.996,Z 1070.649,A -85,B 0,C 180,E1 5212.24,E2 5212.24} C_VEL
LIN {X 0,Y 204.132,Z 1085.213,A -85,B 0,C 180,E1 5209.91,E2 5209.91} C_VEL
LIN {X 0,Y 186.703,Z 1098.653,A -85,B 0,C 180,E1 5207.001,E2 5207.001} C_VEL
LIN {X 0,Y 169.061,Z 1110.551,A -85,B 0,C 180,E1 5203.359,E2 5203.359} C_VEL
LIN {X 0,Y 150.531,Z 1121.64,A -85,B 0,C 180,E1 5198.424,E2 5198.424} C_VEL
LIN {X 0,Y 134.091,Z 1130.401,A -85,B 0,C 180,E1 5192.542,E2 5192.542} C_VEL
LIN {X 0,Y 118.645,Z 1137.755,A -85,B 0,C 180,E1 5184.833,E2 5184.833} C_VEL
LIN {X 0,Y 105.17,Z 1143.778,A -85,B 0,C 180,E1 5174.713,E2 5174.713} C_VEL
LIN {X 0,Y 95.289,Z 1147.932,A -85,B 0,C 180,E1 5162.355,E2 5162.355} C_VEL
LIN {X 0,Y 89.878,Z 1150.527,A -85,B 0,C 180,E1 5148.823,E2 5148.823} C_VEL
LIN {X 0,Y 88.261,Z 1151.487,A -85,B 0,C 180,E1 5137.16,E2 5137.16} C_VEL
LIN {X 0,Y 88.119,Z 1151.657,A -85,B 0,C 180,E1 5128.051,E2 5128.051} C_VEL
LIN {X 0,Y 88.715,Z 1151.17,A -85,B 0,C 180,E1 5117.636,E2 5117.636} C_VEL
LIN {X 0,Y 91.56,Z 1149.638,A -85,B 0,C 180,E1 5105.484,E2 5105.484} C_VEL
LIN {X 0,Y 98.628,Z 1146.607,A -85,B 0,C 180,E1 5092.538,E2 5092.538} C_VEL
LIN {X 0,Y 109.432,Z 1141.909,A -85,B 0,C 180,E1 5081.479,E2 5081.479} C_VEL
LIN {X 0,Y 123.944,Z 1135.413,A -85,B 0,C 180,E1 5072.11,E2 5072.11} C_VEL
LIN {X 0,Y 139.342,Z 1127.77,A -85,B 0,C 180,E1 5065.296,E2 5065.296} C_VEL
LIN {X 0,Y 157.909,Z 1117.499,A -85,B 0,C 180,E1 5059.363,E2 5059.363} C_VEL
LIN {X 0,Y 175.112,Z 1106.787,A -85,B 0,C 180,E1 5055.214,E2 5055.214} C_VEL
LIN {X 0,Y 193.045,Z 1094.069,A -85,B 0,C 180,E1 5051.791,E2 5051.791} C_VEL
LIN {X 0,Y 210.606,Z 1080.082,A -85,B 0,C 180,E1 5049.075,E2 5049.075} C_VEL
LIN {X 0,Y 226.649,Z 1065.427,A -85,B 0,C 180,E1 5046.984,E2 5046.984} C_VEL
LIN {X 0,Y 242.953,Z 1048.663,A -85,B 0,C 180,E1 5045.17,E2 5045.17} C_VEL
LIN {X 0,Y 257.002,Z 1032.118,A -85,B 0,C 180,E1 5043.793,E2 5043.793} C_VEL
LIN {X 0,Y 271.442,Z 1012.679,A -85,B 0,C 180,E1 5042.534,E2 5042.534} C_VEL
LIN {X 0,Y 283.071,Z 994.611,A -85,B 0,C 180,E1 5041.611,E2 5041.611} C_VEL
LIN {X 0,Y 294.444,Z 974.003,A -85,B 0,C 180,E1 5040.779,E2 5040.779} C_VEL
LIN {X 0,Y 300.82,Z 960.728,A -85,B 0,C 180,E1 5040.332,E2 5040.332} C_VEL
LIN {X 0,Y 289.963,Z 982.705,A -85,B 0,C 180,E1 5039.696,E2 5039.696} C_VEL
LIN {X 0,Y 278.833,Z 1001.859,A -85,B 0,C 180,E1 5038.973,E2 5038.973} C_VEL
LIN {X 0,Y 274.968,Z 1007.885,A -85,B 0,C 180,E1 5038.701,E2 5038.701} C_VEL
LIN {X 0,Y 270.562,Z 1014.412,A -85,B 0,C 180,E1 5038.6,E2 5038.6} C_VEL
LIN {X 0,Y 258.541,Z 1030.417,A -85,B 0,C 180,E1 5039.053,E2 5039.053} C_VEL
LIN {X 0,Y 253.719,Z 1036.289,A -85,B 0,C 180,E1 5038.918,E2 5038.918} C_VEL
LIN {X 0,Y 237.186,Z 1055.087,A -85,B 0,C 180,E1 5037.532,E2 5037.532} C_VEL
LIN {X 0,Y 221.51,Z 1070.729,A -85,B 0,C 180,E1 5035.991,E2 5035.991} C_VEL
LIN {X 0,Y 204.102,Z 1086.011,A -85,B 0,C 180,E1 5033.963,E2 5033.963} C_VEL
LIN {X 0,Y 187.007,Z 1099.364,A -85,B 0,C 180,E1 5031.542,E2 5031.542} C_VEL
LIN {X 0,Y 168.489,Z 1112.069,A -85,B 0,C 180,E1 5028.278,E2 5028.278} C_VEL
LIN {X 0,Y 149.789,Z 1123.54,A -85,B 0,C 180,E1 5023.988,E2 5023.988} C_VEL
LIN {X 0,Y 132.126,Z 1133.013,A -85,B 0,C 180,E1 5018.558,E2 5018.558} C_VEL
LIN {X 0,Y 114.513,Z 1141.578,A -85,B 0,C 180,E1 5010.824,E2 5010.824} C_VEL
LIN {X 0,Y 100.681,Z 1147.718,A -85,B 0,C 180,E1 5001.677,E2 5001.677} C_VEL
LIN {X 0,Y 88.605,Z 1152.958,A -85,B 0,C 180,E1 4988.362,E2 4988.362} C_VEL
LIN {X 0,Y 82.465,Z 1155.896,A -85,B 0,C 180,E1 4975.109,E2 4975.109} C_VEL
LIN {X 0,Y 80.142,Z 1157.632,A -85,B 0,C 180,E1 4960.784,E2 4960.784} C_VEL
LIN {X 0,Y 80.108,Z 1158.007,A -85,B 0,C 180,E1 4950.714,E2 4950.714} C_VEL
LIN {X 0,Y 80.081,Z 1157.719,A -85,B 0,C 180,E1 4941.381,E2 4941.381} C_VEL
LIN {X 0,Y 81.875,Z 1156.241,A -85,B 0,C 180,E1 4926.995,E2 4926.995} C_VEL
LIN {X 0,Y 87.824,Z 1153.267,A -85,B 0,C 180,E1 4912.884,E2 4912.884} C_VEL
LIN {X 0,Y 98.926,Z 1148.465,A -85,B 0,C 180,E1 4899.81,E2 4899.81} C_VEL
LIN {X 0,Y 113.088,Z 1142.146,A -85,B 0,C 180,E1 4889.947,E2 4889.947} C_VEL
LIN {X 0,Y 131.317,Z 1133.345,A -85,B 0,C 180,E1 4881.73,E2 4881.73} C_VEL
LIN {X 0,Y 148.922,Z 1123.919,A -85,B 0,C 180,E1 4876.235,E2 4876.235} C_VEL
LIN {X 0,Y 167.58,Z 1112.534,A -85,B 0,C 180,E1 4871.898,E2 4871.898} C_VEL
LIN {X 0,Y 186.068,Z 1099.921,A -85,B 0,C 180,E1 4868.597,E2 4868.597} C_VEL
LIN {X 0,Y 203.144,Z 1086.617,A -85,B 0,C 180,E1 4866.15,E2 4866.15} C_VEL
LIN {X 0,Y 220.538,Z 1071.45,A -85,B 0,C 180,E1 4864.104,E2 4864.104} C_VEL
LIN {X 0,Y 236.204,Z 1055.871,A -85,B 0,C 180,E1 4862.546,E2 4862.546} C_VEL
LIN {X 0,Y 253.017,Z 1036.862,A -85,B 0,C 180,E1 4861.126,E2 4861.126} C_VEL
LIN {X 0,Y 266.967,Z 1018.769,A -85,B 0,C 180,E1 4860.107,E2 4860.107} C_VEL
LIN {X 0,Y 276.501,Z 1004.856,A -85,B 0,C 180,E1 4859.485,E2 4859.485} C_VEL
LIN {X 0,Y 263.555,Z 1023.165,A -85,B 0,C 180,E1 4858.512,E2 4858.512} C_VEL
LIN {X 0,Y 249.244,Z 1040.987,A -85,B 0,C 180,E1 4857.307,E2 4857.307} C_VEL
LIN {X 0,Y 234.565,Z 1056.869,A -85,B 0,C 180,E1 4855.921,E2 4855.921} C_VEL
LIN {X 0,Y 218.116,Z 1072.66,A -85,B 0,C 180,E1 4854.131,E2 4854.131} C_VEL
LIN {X 0,Y 201.555,Z 1086.565,A -85,B 0,C 180,E1 4852.015,E2 4852.015} C_VEL
LIN {X 0,Y 182.311,Z 1100.796,A -85,B 0,C 180,E1 4849.027,E2 4849.027} C_VEL
LIN {X 0,Y 164.546,Z 1112.335,A -85,B 0,C 180,E1 4845.573,E2 4845.573} C_VEL
LIN {X 0,Y 145.997,Z 1122.845,A -85,B 0,C 180,E1 4840.929,E2 4840.929} C_VEL
LIN {X 0,Y 128.135,Z 1131.853,A -85,B 0,C 180,E1 4834.849,E2 4834.849} C_VEL
LIN {X 0,Y 111.856,Z 1139.009,A -85,B 0,C 180,E1 4826.956,E2 4826.956} C_VEL
LIN {X 0,Y 96.736,Z 1145.08,A -85,B 0,C 180,E1 4815.497,E2 4815.497} C_VEL
LIN {X 0,Y 87.365,Z 1148.693,A -85,B 0,C 180,E1 4803.324,E2 4803.324} C_VEL
LIN {X 0,Y 81.575,Z 1151.078,A -85,B 0,C 180,E1 4787.846,E2 4787.846} C_VEL
LIN {X 0,Y 80.229,Z 1151.827,A -85,B 0,C 180,E1 4776.442,E2 4776.442} C_VEL
LIN {X 0,Y 80.13,Z 1151.936,A -85,B 0,C 180,E1 4767.141,E2 4767.141} C_VEL
LIN {X 0,Y 80.937,Z 1151.41,A -85,B 0,C 180,E1 4755.697,E2 4755.697} C_VEL
LIN {X 0,Y 84.478,Z 1149.837,A -85,B 0,C 180,E1 4742.511,E2 4742.511} C_VEL
LIN {X 0,Y 93.173,Z 1146.521,A -85,B 0,C 180,E1 4728.293,E2 4728.293} C_VEL
LIN {X 0,Y 104.76,Z 1141.975,A -85,B 0,C 180,E1 4717.612,E2 4717.612} C_VEL
LIN {X 0,Y 121.257,Z 1135.023,A -85,B 0,C 180,E1 4708.036,E2 4708.036} C_VEL
LIN {X 0,Y 137.638,Z 1127.292,A -85,B 0,C 180,E1 4701.591,E2 4701.591} C_VEL
LIN {X 0,Y 156.231,Z 1117.304,A -85,B 0,C 180,E1 4696.266,E2 4696.266} C_VEL
LIN {X 0,Y 174.037,Z 1106.534,A -85,B 0,C 180,E1 4692.403,E2 4692.403} C_VEL
LIN {X 0,Y 192.159,Z 1093.914,A -85,B 0,C 180,E1 4689.283,E2 4689.283} C_VEL
LIN {X 0,Y 209.506,Z 1080.354,A -85,B 0,C 180,E1 4686.853,E2 4686.853} C_VEL
LIN {X 0,Y 225.801,Z 1065.731,A -85,B 0,C 180,E1 4684.924,E2 4684.924} C_VEL
LIN {X 0,Y 242.355,Z 1048.965,A -85,B 0,C 180,E1 4683.25,E2 4683.25} C_VEL
LIN {X 0,Y 256.616,Z 1032.39,A -85,B 0,C 180,E1 4681.981,E2 4681.981} C_VEL
LIN {X 0,Y 271.488,Z 1012.564,A -85,B 0,C 180,E1 4680.804,E2 4680.804} C_VEL
LIN {X 0,Y 275.97,Z 1006.009,A -85,B 0,C 180,E1 4680.469,E2 4680.469} C_VEL
LIN {X 0,Y 262.969,Z 1024.494,A -85,B 0,C 180,E1 4679.604,E2 4679.604} C_VEL
LIN {X 0,Y 253.719,Z 1036.289,A -85,B 0,C 180,E1 4678.918,E2 4678.918} C_VEL
LIN {X 0,Y 248.735,Z 1042.234,A -85,B 0,C 180,E1 4678.763,E2 4678.763} C_VEL
LIN {X 0,Y 235.062,Z 1056.906,A -85,B 0,C 180,E1 4679.12,E2 4679.12} C_VEL
LIN {X 0,Y 229.611,Z 1062.347,A -85,B 0,C 180,E1 4678.907,E2 4678.907} C_VEL
LIN {X 0,Y 212.213,Z 1078.314,A -85,B 0,C 180,E1 4677.255,E2 4677.255} C_VEL
LIN {X 0,Y 193.675,Z 1093.35,A -85,B 0,C 180,E1 4675.115,E2 4675.115} C_VEL
LIN {X 0,Y 176.417,Z 1105.636,A -85,B 0,C 180,E1 4672.667,E2 4672.667} C_VEL
LIN {X 0,Y 155.613,Z 1118.657,A -85,B 0,C 180,E1 4668.887,E2 4668.887} C_VEL
LIN {X 0,Y 136.866,Z 1128.98,A -85,B 0,C 180,E1 4664.319,E2 4664.319} C_VEL
LIN {X 0,Y 118.529,Z 1137.76,A -85,B 0,C 180,E1 4658.109,E2 4658.109} C_VEL
LIN {X 0,Y 101.83,Z 1145.012,A -85,B 0,C 180,E1 4649.774,E2 4649.774} C_VEL
LIN {X 0,Y 87.856,Z 1150.468,A -85,B 0,C 180,E1 4638.686,E2 4638.686} C_VEL
LIN {X 0,Y 77.458,Z 1154.603,A -85,B 0,C 180,E1 4623.713,E2 4623.713} C_VEL
LIN {X 0,Y 72.858,Z 1156.736,A -85,B 0,C 180,E1 4608.398,E2 4608.398} C_VEL
LIN {X 0,Y 72.064,Z 1157.53,A -85,B 0,C 180,E1 4596.371,E2 4596.371} C_VEL
LIN {X 0,Y 72.091,Z 1157.655,A -85,B 0,C 180,E1 4587.614,E2 4587.614} C_VEL
LIN {X 0,Y 72.306,Z 1157.174,A -85,B 0,C 180,E1 4576.402,E2 4576.402} C_VEL
LIN {X 0,Y 75.592,Z 1155.335,A -85,B 0,C 180,E1 4560.804,E2 4560.804} C_VEL
LIN {X 0,Y 84.255,Z 1151.901,A -85,B 0,C 180,E1 4545.398,E2 4545.398} C_VEL
LIN {X 0,Y 97.7,Z 1146.556,A -85,B 0,C 180,E1 4532.943,E2 4532.943} C_VEL
LIN {X 0,Y 114.547,Z 1139.511,A -85,B 0,C 180,E1 4523.573,E2 4523.573} C_VEL
LIN {X 0,Y 131.856,Z 1131.361,A -85,B 0,C 180,E1 4517.162,E2 4517.162} C_VEL
LIN {X 0,Y 152.218,Z 1120.508,A -85,B 0,C 180,E1 4511.835,E2 4511.835} C_VEL
LIN {X 0,Y 170.748,Z 1109.289,A -85,B 0,C 180,E1 4508.253,E2 4508.253} C_VEL
LIN {X 0,Y 189.813,Z 1096.04,A -85,B 0,C 180,E1 4505.381,E2 4505.381} C_VEL
LIN {X 0,Y 208.29,Z 1081.543,A -85,B 0,C 180,E1 4503.158,E2 4503.158} C_VEL
LIN {X 0,Y 225.048,Z 1066.446,A -85,B 0,C 180,E1 4501.491,E2 4501.491} C_VEL
LIN {X 0,Y 241.97,Z 1049.214,A -85,B 0,C 180,E1 4500.075,E2 4500.075} C_VEL
LIN {X 0,Y 251.45,Z 1038.435,A -85,B 0,C 180,E1 4499.373,E2 4499.373} C_VEL
LIN {X 0,Y 235.696,Z 1055.586,A -85,B 0,C 180,E1 4498.055,E2 4498.055} C_VEL
LIN {X 0,Y 219.387,Z 1071.269,A -85,B 0,C 180,E1 4496.48,E2 4496.48} C_VEL
LIN {X 0,Y 201.903,Z 1085.834,A -85,B 0,C 180,E1 4494.505,E2 4494.505} C_VEL
LIN {X 0,Y 183.755,Z 1099.238,A -85,B 0,C 180,E1 4492.024,E2 4492.024} C_VEL
LIN {X 0,Y 165.09,Z 1111.175,A -85,B 0,C 180,E1 4488.861,E2 4488.861} C_VEL
LIN {X 0,Y 144.748,Z 1122.526,A -85,B 0,C 180,E1 4484.371,E2 4484.371} C_VEL
LIN {X 0,Y 126.484,Z 1131.418,A -85,B 0,C 180,E1 4478.878,E2 4478.878} C_VEL
LIN {X 0,Y 109.207,Z 1138.67,A -85,B 0,C 180,E1 4471.518,E2 4471.518} C_VEL
LIN {X 0,Y 93.551,Z 1144.603,A -85,B 0,C 180,E1 4461.283,E2 4461.283} C_VEL
LIN {X 0,Y 81.909,Z 1148.548,A -85,B 0,C 180,E1 4448.505,E2 4448.505} C_VEL
LIN {X 0,Y 74.683,Z 1151.137,A -85,B 0,C 180,E1 4432.848,E2 4432.848} C_VEL
LIN {X 0,Y 72.351,Z 1152.089,A -85,B 0,C 180,E1 4418.746,E2 4418.746} C_VEL
LIN {X 0,Y 72.132,Z 1152.257,A -85,B 0,C 180,E1 4407.618,E2 4407.618} C_VEL
LIN {X 0,Y 73.01,Z 1151.776,A -85,B 0,C 180,E1 4394.92,E2 4394.92} C_VEL
LIN {X 0,Y 77.014,Z 1150.249,A -85,B 0,C 180,E1 4380.441,E2 4380.441} C_VEL
LIN {X 0,Y 86.159,Z 1147.223,A -85,B 0,C 180,E1 4365.872,E2 4365.872} C_VEL
LIN {X 0,Y 99.258,Z 1142.528,A -85,B 0,C 180,E1 4354.31,E2 4354.31} C_VEL
LIN {X 0,Y 115.994,Z 1136.031,A -85,B 0,C 180,E1 4345.166,E2 4345.166} C_VEL
LIN {X 0,Y 133.111,Z 1128.389,A -85,B 0,C 180,E1 4338.838,E2 4338.838} C_VEL
LIN {X 0,Y 153.22,Z 1118.116,A -85,B 0,C 180,E1 4333.514,E2 4333.514} C_VEL
LIN {X 0,Y 171.521,Z 1107.403,A -85,B 0,C 180,E1 4329.885,E2 4329.885} C_VEL
LIN {X 0,Y 190.365,Z 1094.682,A -85,B 0,C 180,E1 4326.936,E2 4326.936} C_VEL
LIN {X 0,Y 208.648,Z 1080.692,A -85,B 0,C 180,E1 4324.62,E2 4324.62} C_VEL
LIN {X 0,Y 225.246,Z 1066.035,A -85,B 0,C 180,E1 4322.851,E2 4322.851} C_VEL
LIN {X 0,Y 242.03,Z 1049.267,A -85,B 0,C 180,E1 4321.323,E2 4321.323} C_VEL
LIN {X 0,Y 250.977,Z 1039.314,A -85,B 0,C 180,E1 4320.581,E2 4320.581} C_VEL
LIN {X 0,Y 234.981,Z 1056.832,A -85,B 0,C 180,E1 4319.364,E2 4319.364} C_VEL
LIN {X 0,Y 229.611,Z 1062.347,A -85,B 0,C 180,E1 4318.907,E2 4318.907} C_VEL
LIN {X 0,Y 224.018,Z 1067.654,A -85,B 0,C 180,E1 4318.67,E2 4318.67} C_VEL
LIN {X 0,Y 207.927,Z 1081.535,A -85,B 0,C 180,E1 4318.892,E2 4318.892} C_VEL
LIN {X 0,Y 202.796,Z 1085.577,A -85,B 0,C 180,E1 4318.608,E2 4318.608} C_VEL
LIN {X 0,Y 184.311,Z 1099.456,A -85,B 0,C 180,E1 4316.527,E2 4316.527} C_VEL
LIN {X 0,Y 164.942,Z 1112.031,A -85,B 0,C 180,E1 4313.795,E2 4313.795} C_VEL
LIN {X 0,Y 145.125,Z 1123.385,A -85,B 0,C 180,E1 4310.134,E2 4310.134} C_VEL
LIN {X 0,Y 126.069,Z 1132.803,A -85,B 0,C 180,E1 4305.369,E2 4305.369} C_VEL
LIN {X 0,Y 105.717,Z 1141.581,A -85,B 0,C 180,E1 4297.951,E2 4297.951} C_VEL
LIN {X 0,Y 89.153,Z 1147.89,A -85,B 0,C 180,E1 4288.466,E2 4288.466} C_VEL
LIN {X 0,Y 75.245,Z 1152.676,A -85,B 0,C 180,E1 4274.768,E2 4274.768} C_VEL
LIN {X 0,Y 67.012,Z 1155.672,A -85,B 0,C 180,E1 4258.323,E2 4258.323} C_VEL
LIN {X 0,Y 64.144,Z 1157.117,A -85,B 0,C 180,E1 4240.779,E2 4240.779} C_VEL
LIN {X 0,Y 64.127,Z 1157.422,A -85,B 0,C 180,E1 4229.998,E2 4229.998} C_VEL
LIN {X 0,Y 64.148,Z 1157.108,A -85,B 0,C 180,E1 4219.09,E2 4219.09} C_VEL
LIN {X 0,Y 67.341,Z 1155.502,A -85,B 0,C 180,E1 4200.659,E2 4200.659} C_VEL
LIN {X 0,Y 75.245,Z 1152.643,A -85,B 0,C 180,E1 4185.227,E2 4185.227} C_VEL
LIN {X 0,Y 89.153,Z 1147.837,A -85,B 0,C 180,E1 4171.529,E2 4171.529} C_VEL
LIN {X 0,Y 105.718,Z 1141.515,A -85,B 0,C 180,E1 4162.045,E2 4162.045} C_VEL
LIN {X 0,Y 126.07,Z 1132.713,A -85,B 0,C 180,E1 4154.625,E2 4154.625} C_VEL
LIN {X 0,Y 145.126,Z 1123.286,A -85,B 0,C 180,E1 4149.86,E2 4149.86} C_VEL
LIN {X 0,Y 164.944,Z 1111.903,A -85,B 0,C 180,E1 4146.198,E2 4146.198} C_VEL
LIN {X 0,Y 184.721,Z 1098.994,A -85,B 0,C 180,E1 4143.413,E2 4143.413} C_VEL
LIN {X 0,Y 202.487,Z 1085.637,A -85,B 0,C 180,E1 4141.414,E2 4141.414} C_VEL
LIN {X 0,Y 220.975,Z 1069.885,A -85,B 0,C 180,E1 4139.714,E2 4139.714} C_VEL
LIN {X 0,Y 226.368,Z 1064.84,A -85,B 0,C 180,E1 4139.272,E2 4139.272} C_VEL
LIN {X 0,Y 210.134,Z 1079.108,A -85,B 0,C 180,E1 4137.76,E2 4137.76} C_VEL
LIN {X 0,Y 191.516,Z 1093.424,A -85,B 0,C 180,E1 4135.697,E2 4135.697} C_VEL
LIN {X 0,Y 173.193,Z 1105.778,A -85,B 0,C 180,E1 4133.213,E2 4133.213} C_VEL
LIN {X 0,Y 153.702,Z 1117.114,A -85,B 0,C 180,E1 4129.883,E2 4129.883} C_VEL
LIN {X 0,Y 134.269,Z 1127.009,A -85,B 0,C 180,E1 4125.487,E2 4125.487} C_VEL
LIN {X 0,Y 115.256,Z 1135.211,A -85,B 0,C 180,E1 4119.543,E2 4119.543} C_VEL
LIN {X 0,Y 96.355,Z 1142.274,A -85,B 0,C 180,E1 4110.654,E2 4110.654} C_VEL
LIN {X 0,Y 82.033,Z 1146.953,A -85,B 0,C 180,E1 4099.758,E2 4099.758} C_VEL
LIN {X 0,Y 70.432,Z 1150.414,A -85,B 0,C 180,E1 4083.62,E2 4083.62} C_VEL
LIN {X 0,Y 65.396,Z 1151.995,A -85,B 0,C 180,E1 4067.808,E2 4067.808} C_VEL
LIN {X 0,Y 64.16,Z 1152.516,A -85,B 0,C 180,E1 4054.135,E2 4054.135} C_VEL
LIN {X 0,Y 64.218,Z 1152.475,A -85,B 0,C 180,E1 4043.745,E2 4043.745} C_VEL
LIN {X 0,Y 65.718,Z 1151.892,A -85,B 0,C 180,E1 4030.447,E2 4030.447} C_VEL
LIN {X 0,Y 71.569,Z 1150.133,A -85,B 0,C 180,E1 4014.074,E2 4014.074} C_VEL
LIN {X 0,Y 83.421,Z 1146.547,A -85,B 0,C 180,E1 3998.827,E2 3998.827} C_VEL
LIN {X 0,Y 98.534,Z 1141.618,A -85,B 0,C 180,E1 3988.017,E2 3988.017} C_VEL
LIN {X 0,Y 116.039,Z 1134.973,A -85,B 0,C 180,E1 3980.084,E2 3980.084} C_VEL
LIN {X 0,Y 135.114,Z 1126.72,A -85,B 0,C 180,E1 3974.209,E2 3974.209} C_VEL
LIN {X 0,Y 154.286,Z 1116.916,A -85,B 0,C 180,E1 3969.925,E2 3969.925} C_VEL
LIN {X 0,Y 174.117,Z 1105.325,A -85,B 0,C 180,E1 3966.568,E2 3966.568} C_VEL
LIN {X 0,Y 191.826,Z 1093.376,A -85,B 0,C 180,E1 3964.185,E2 3964.185} C_VEL
LIN {X 0,Y 211.106,Z 1078.499,A -85,B 0,C 180,E1 3962.063,E2 3962.063} C_VEL
LIN {X 0,Y 225.927,Z 1065.477,A -85,B 0,C 180,E1 3960.683,E2 3960.683} C_VEL
LIN {X 0,Y 208.603,Z 1080.911,A -85,B 0,C 180,E1 3959.177,E2 3959.177} C_VEL
LIN {X 0,Y 202.796,Z 1085.577,A -85,B 0,C 180,E1 3958.608,E2 3958.608} C_VEL
LIN {X 0,Y 196.682,Z 1090.365,A -85,B 0,C 180,E1 3958.278,E2 3958.278} C_VEL
LIN {X 0,Y 180.133,Z 1101.773,A -85,B 0,C 180,E1 3958.367,E2 3958.367} C_VEL
LIN {X 0,Y 173.752,Z 1105.878,A -85,B 0,C 180,E1 3957.939,E2 3957.939} C_VEL
LIN {X 0,Y 153.541,Z 1117.883,A -85,B 0,C 180,E1 3955.088,E2 3955.088} C_VEL
LIN {X 0,Y 133.507,Z 1128.256,A -85,B 0,C 180,E1 3951.324,E2 3951.324} C_VEL
LIN {X 0,Y 113.344,Z 1137.132,A -85,B 0,C 180,E1 3946.011,E2 3946.011} C_VEL
LIN {X 0,Y 94.507,Z 1144.385,A -85,B 0,C 180,E1 3938.591,E2 3938.591} C_VEL
LIN {X 0,Y 77.847,Z 1149.843,A -85,B 0,C 180,E1 3927.96,E2 3927.96} C_VEL
LIN {X 0,Y 64.356,Z 1153.984,A -85,B 0,C 180,E1 3911.915,E2 3911.915} C_VEL
LIN {X 0,Y 57.576,Z 1156.123,A -85,B 0,C 180,E1 3893.54,E2 3893.54} C_VEL
LIN {X 0,Y 56.077,Z 1156.926,A -85,B 0,C 180,E1 3878.198,E2 3878.198} C_VEL
LIN {X 0,Y 56.103,Z 1157.079,A -85,B 0,C 180,E1 3867.955,E2 3867.955} C_VEL
LIN {X 0,Y 56.519,Z 1156.639,A -85,B 0,C 180,E1 3853.555,E2 3853.555} C_VEL
LIN {X 0,Y 61.371,Z 1154.823,A -85,B 0,C 180,E1 3834.088,E2 3834.088} C_VEL
LIN {X 0,Y 71.981,Z 1151.649,A -85,B 0,C 180,E1 3817.646,E2 3817.646} C_VEL
LIN {X 0,Y 88.178,Z 1146.445,A -85,B 0,C 180,E1 3804.804,E2 3804.804} C_VEL
LIN {X 0,Y 107.178,Z 1139.608,A -85,B 0,C 180,E1 3796.073,E2 3796.073} C_VEL
LIN {X 0,Y 126.985,Z 1131.145,A -85,B 0,C 180,E1 3790.181,E2 3790.181} C_VEL
LIN {X 0,Y 148.129,Z 1120.727,A -85,B 0,C 180,E1 3785.81,E2 3785.81} C_VEL
LIN {X 0,Y 167.194,Z 1109.83,A -85,B 0,C 180,E1 3782.899,E2 3782.899} C_VEL
LIN {X 0,Y 187.983,Z 1096.124,A -85,B 0,C 180,E1 3780.445,E2 3780.445} C_VEL
LIN {X 0,Y 200.996,Z 1086.454,A -85,B 0,C 180,E1 3779.167,E2 3779.167} C_VEL
LIN {X 0,Y 182.201,Z 1099.86,A -85,B 0,C 180,E1 3777.16,E2 3777.16} C_VEL
LIN {X 0,Y 162.709,Z 1111.797,A -85,B 0,C 180,E1 3774.577,E2 3774.577} C_VEL
LIN {X 0,Y 141.745,Z 1122.886,A -85,B 0,C 180,E1 3770.957,E2 3770.957} C_VEL
LIN {X 0,Y 122.403,Z 1131.648,A -85,B 0,C 180,E1 3766.43,E2 3766.43} C_VEL
LIN {X 0,Y 103.195,Z 1139,A -85,B 0,C 180,E1 3760.029,E2 3760.029} C_VEL
LIN {X 0,Y 84.957,Z 1145.018,A -85,B 0,C 180,E1 3750.568,E2 3750.568} C_VEL
LIN {X 0,Y 69.82,Z 1149.164,A -85,B 0,C 180,E1 3736.919,E2 3736.919} C_VEL
LIN {X 0,Y 60.025,Z 1151.747,A -85,B 0,C 180,E1 3718.889,E2 3718.889} C_VEL
LIN {X 0,Y 56.433,Z 1152.711,A -85,B 0,C 180,E1 3700.208,E2 3700.208} C_VEL
LIN {X 0,Y 56.139,Z 1152.878,A -85,B 0,C 180,E1 3687.961,E2 3687.961} C_VEL
LIN {X 0,Y 57.215,Z 1152.506,A -85,B 0,C 180,E1 3672.72,E2 3672.72} C_VEL
LIN {X 0,Y 62.903,Z 1150.966,A -85,B 0,C 180,E1 3653.978,E2 3653.978} C_VEL
LIN {X 0,Y 74.578,Z 1148.009,A -85,B 0,C 180,E1 3637.723,E2 3637.723} C_VEL
LIN {X 0,Y 90.97,Z 1143.146,A -85,B 0,C 180,E1 3625.677,E2 3625.677} C_VEL
LIN {X 0,Y 109.978,Z 1136.65,A -85,B 0,C 180,E1 3617.333,E2 3617.333} C_VEL
LIN {X 0,Y 128.721,Z 1129.007,A -85,B 0,C 180,E1 3611.844,E2 3611.844} C_VEL
LIN {X 0,Y 150.219,Z 1118.733,A -85,B 0,C 180,E1 3607.37,E2 3607.37} C_VEL
LIN {X 0,Y 169.47,Z 1108.018,A -85,B 0,C 180,E1 3604.381,E2 3604.381} C_VEL
LIN {X 0,Y 189.085,Z 1095.295,A -85,B 0,C 180,E1 3601.979,E2 3601.979} C_VEL
LIN {X 0,Y 200.746,Z 1086.84,A -85,B 0,C 180,E1 3600.777,E2 3600.777} C_VEL
LIN {X 0,Y 182.007,Z 1100.483,A -85,B 0,C 180,E1 3598.902,E2 3598.902} C_VEL
LIN {X 0,Y 173.752,Z 1105.878,A -85,B 0,C 180,E1 3597.939,E2 3597.939} C_VEL
LIN {X 0,Y 167.274,Z 1109.931,A -85,B 0,C 180,E1 3597.464,E2 3597.464} C_VEL
LIN {X 0,Y 149.613,Z 1119.597,A -85,B 0,C 180,E1 3597.322,E2 3597.322} C_VEL
LIN {X 0,Y 142.799,Z 1122.955,A -85,B 0,C 180,E1 3596.697,E2 3596.697} C_VEL
LIN {X 0,Y 122.907,Z 1132.176,A -85,B 0,C 180,E1 3592.964,E2 3592.964} C_VEL
LIN {X 0,Y 100.376,Z 1141.041,A -85,B 0,C 180,E1 3586.757,E2 3586.757} C_VEL
LIN {X 0,Y 81.384,Z 1147.352,A -85,B 0,C 180,E1 3578.374,E2 3578.374} C_VEL
LIN {X 0,Y 64.512,Z 1152.053,A -85,B 0,C 180,E1 3565.226,E2 3565.226} C_VEL
LIN {X 0,Y 52.781,Z 1155.154,A -85,B 0,C 180,E1 3545.959,E2 3545.959} C_VEL
LIN {X 0,Y 48.232,Z 1156.542,A -85,B 0,C 180,E1 3523.025,E2 3523.025} C_VEL
LIN {X 0,Y 48.134,Z 1156.822,A -85,B 0,C 180,E1 3509.997,E2 3509.997} C_VEL
LIN {X 0,Y 48.312,Z 1156.504,A -85,B 0,C 180,E1 3495.617,E2 3495.617} C_VEL
LIN {X 0,Y 53.58,Z 1154.882,A -85,B 0,C 180,E1 3471.986,E2 3471.986} C_VEL
LIN {X 0,Y 65.176,Z 1151.848,A -85,B 0,C 180,E1 3454.061,E2 3454.061} C_VEL
LIN {X 0,Y 84.128,Z 1146.41,A -85,B 0,C 180,E1 3440.125,E2 3440.125} C_VEL
LIN {X 0,Y 103.341,Z 1139.938,A -85,B 0,C 180,E1 3432.25,E2 3432.25} C_VEL
LIN {X 0,Y 123.862,Z 1131.664,A -85,B 0,C 180,E1 3426.821,E2 3426.821} C_VEL
LIN {X 0,Y 144.191,Z 1122.181,A -85,B 0,C 180,E1 3423.079,E2 3423.079} C_VEL
LIN {X 0,Y 164.982,Z 1110.686,A -85,B 0,C 180,E1 3420.263,E2 3420.263} C_VEL
LIN {X 0,Y 175.467,Z 1104.242,A -85,B 0,C 180,E1 3419.065,E2 3419.065} C_VEL
LIN {X 0,Y 154.283,Z 1116.394,A -85,B 0,C 180,E1 3416.414,E2 3416.414} C_VEL
LIN {X 0,Y 134.919,Z 1125.879,A -85,B 0,C 180,E1 3413.251,E2 3413.251} C_VEL
LIN {X 0,Y 113.313,Z 1134.808,A -85,B 0,C 180,E1 3408.372,E2 3408.372} C_VEL
LIN {X 0,Y 92.827,Z 1141.92,A -85,B 0,C 180,E1 3401.423,E2 3401.423} C_VEL
LIN {X 0,Y 75,Z 1146.908,A -85,B 0,C 180,E1 3391.631,E2 3391.631} C_VEL
LIN {X 0,Y 59.679,Z 1150.608,A -85,B 0,C 180,E1 3376.092,E2 3376.092} C_VEL
LIN {X 0,Y 50.75,Z 1152.48,A -85,B 0,C 180,E1 3355.689,E2 3355.689} C_VEL
LIN {X 0,Y 48.308,Z 1153.07,A -85,B 0,C 180,E1 3338.333,E2 3338.333} C_VEL
LIN {X 0,Y 48.183,Z 1153.131,A -85,B 0,C 180,E1 3324.936,E2 3324.936} C_VEL
LIN {X 0,Y 49.975,Z 1152.685,A -85,B 0,C 180,E1 3307.66,E2 3307.66} C_VEL
LIN {X 0,Y 56.993,Z 1151.167,A -85,B 0,C 180,E1 3288.194,E2 3288.194} C_VEL
LIN {X 0,Y 71.27,Z 1147.951,A -85,B 0,C 180,E1 3271.156,E2 3271.156} C_VEL
LIN {X 0,Y 88.544,Z 1143.211,A -85,B 0,C 180,E1 3260.408,E2 3260.408} C_VEL
LIN {X 0,Y 109.618,Z 1136.276,A -85,B 0,C 180,E1 3252.588,E2 3252.588} C_VEL
LIN {X 0,Y 129.175,Z 1128.529,A -85,B 0,C 180,E1 3247.797,E2 3247.797} C_VEL
LIN {X 0,Y 150.358,Z 1118.538,A -85,B 0,C 180,E1 3244.078,E2 3244.078} C_VEL
LIN {X 0,Y 170.031,Z 1107.764,A -85,B 0,C 180,E1 3241.478,E2 3241.478} C_VEL
LIN {X 0,Y 175.332,Z 1104.484,A -85,B 0,C 180,E1 3240.871,E2 3240.871} C_VEL
LIN {X 0,Y 153.051,Z 1117.57,A -85,B 0,C 180,E1 3238.215,E2 3238.215} C_VEL
LIN {X 0,Y 142.799,Z 1122.955,A -85,B 0,C 180,E1 3236.697,E2 3236.697} C_VEL
LIN {X 0,Y 135.922,Z 1126.211,A -85,B 0,C 180,E1 3235.997,E2 3235.997} C_VEL
LIN {X 0,Y 116.341,Z 1134.349,A -85,B 0,C 180,E1 3235.359,E2 3235.359} C_VEL
LIN {X 0,Y 110.351,Z 1136.558,A -85,B 0,C 180,E1 3234.466,E2 3234.466} C_VEL
LIN {X 0,Y 88.838,Z 1144.024,A -85,B 0,C 180,E1 3228.281,E2 3228.281} C_VEL
LIN {X 0,Y 69.319,Z 1149.508,A -85,B 0,C 180,E1 3218.865,E2 3218.865} C_VEL
LIN {X 0,Y 51.299,Z 1153.734,A -85,B 0,C 180,E1 3201.224,E2 3201.224} C_VEL
LIN {X 0,Y 42.213,Z 1155.712,A -85,B 0,C 180,E1 3178.797,E2 3178.797} C_VEL
LIN {X 0,Y 40.08,Z 1156.431,A -85,B 0,C 180,E1 3155.724,E2 3155.724} C_VEL
LIN {X 0,Y 40.085,Z 1156.452,A -85,B 0,C 180,E1 3145.705,E2 3145.705} C_VEL
LIN {X 0,Y 41.845,Z 1155.799,A -85,B 0,C 180,E1 3122.996,E2 3122.996} C_VEL
LIN {X 0,Y 50.105,Z 1153.956,A -85,B 0,C 180,E1 3100.681,E2 3100.681} C_VEL
LIN {X 0,Y 66.609,Z 1150.188,A -85,B 0,C 180,E1 3082.97,E2 3082.97} C_VEL
LIN {X 0,Y 85.206,Z 1145.03,A -85,B 0,C 180,E1 3073.093,E2 3073.093} C_VEL
LIN {X 0,Y 107.612,Z 1137.516,A -85,B 0,C 180,E1 3066.173,E2 3066.173} C_VEL
LIN {X 0,Y 128.07,Z 1129.261,A -85,B 0,C 180,E1 3062.088,E2 3062.088} C_VEL
LIN {X 0,Y 150.005,Z 1118.717,A -85,B 0,C 180,E1 3058.993,E2 3058.993} C_VEL
LIN {X 0,Y 128.331,Z 1128.731,A -85,B 0,C 180,E1 3055.791,E2 3055.791} C_VEL
LIN {X 0,Y 108.141,Z 1136.488,A -85,B 0,C 180,E1 3051.624,E2 3051.624} C_VEL
LIN {X 0,Y 86.044,Z 1143.45,A -85,B 0,C 180,E1 3044.692,E2 3044.692} C_VEL
LIN {X 0,Y 67.414,Z 1148.201,A -85,B 0,C 180,E1 3034.792,E2 3034.792} C_VEL
LIN {X 0,Y 51.216,Z 1151.44,A -85,B 0,C 180,E1 3017.893,E2 3017.893} C_VEL
LIN {X 0,Y 42.326,Z 1153.031,A -85,B 0,C 180,E1 2995.168,E2 2995.168} C_VEL
LIN {X 0,Y 40.173,Z 1153.45,A -85,B 0,C 180,E1 2974.285,E2 2974.285} C_VEL
LIN {X 0,Y 40.469,Z 1153.358,A -85,B 0,C 180,E1 2958.603,E2 2958.603} C_VEL
LIN {X 0,Y 44.284,Z 1152.682,A -85,B 0,C 180,E1 2937.191,E2 2937.191} C_VEL
LIN {X 0,Y 56.956,Z 1150.429,A -85,B 0,C 180,E1 2914.407,E2 2914.407} C_VEL
LIN {X 0,Y 73.904,Z 1146.686,A -85,B 0,C 180,E1 2901.015,E2 2901.015} C_VEL
LIN {X 0,Y 95.974,Z 1140.583,A -85,B 0,C 180,E1 2891.685,E2 2891.685} C_VEL
LIN {X 0,Y 116.699,Z 1133.507,A -85,B 0,C 180,E1 2886.352,E2 2886.352} C_VEL
LIN {X 0,Y 138.117,Z 1124.521,A -85,B 0,C 180,E1 2882.558,E2 2882.558} C_VEL
LIN {X 0,Y 149.694,Z 1119,A -85,B 0,C 180,E1 2880.961,E2 2880.961} C_VEL
LIN {X 0,Y 127.079,Z 1129.775,A -85,B 0,C 180,E1 2877.744,E2 2877.744} C_VEL
LIN {X 0,Y 110.351,Z 1136.558,A -85,B 0,C 180,E1 2874.466,E2 2874.466} C_VEL
LIN {X 0,Y 103.298,Z 1139.145,A -85,B 0,C 180,E1 2873.346,E2 2873.346} C_VEL
LIN {X 0,Y 83.586,Z 1144.887,A -85,B 0,C 180,E1 2871.796,E2 2871.796} C_VEL
LIN {X 0,Y 76.998,Z 1146.67,A -85,B 0,C 180,E1 2870.145,E2 2870.145} C_VEL
LIN {X 0,Y 56.688,Z 1151.43,A -85,B 0,C 180,E1 2859.192,E2 2859.192} C_VEL
LIN {X 0,Y 40.005,Z 1154.653,A -85,B 0,C 180,E1 2838.569,E2 2838.569} C_VEL
LIN {X 0,Y 32.432,Z 1155.972,A -85,B 0,C 180,E1 2807.128,E2 2807.128} C_VEL
LIN {X 0,Y 32.138,Z 1156.222,A -85,B 0,C 180,E1 2789.996,E2 2789.996} C_VEL
LIN {X 0,Y 32.82,Z 1155.895,A -85,B 0,C 180,E1 2768.552,E2 2768.552} C_VEL
LIN {X 0,Y 41.827,Z 1154.263,A -85,B 0,C 180,E1 2737.916,E2 2737.916} C_VEL
LIN {X 0,Y 57.525,Z 1151.222,A -85,B 0,C 180,E1 2720.176,E2 2720.176} C_VEL
LIN {X 0,Y 79.926,Z 1145.779,A -85,B 0,C 180,E1 2708.768,E2 2708.768} C_VEL
LIN {X 0,Y 101.553,Z 1139.167,A -85,B 0,C 180,E1 2702.82,E2 2702.82} C_VEL
LIN {X 0,Y 123.901,Z 1130.659,A -85,B 0,C 180,E1 2698.901,E2 2698.901} C_VEL
LIN {X 0,Y 102.234,Z 1138.518,A -85,B 0,C 180,E1 2694.949,E2 2694.949} C_VEL
LIN {X 0,Y 81.44,Z 1144.492,A -85,B 0,C 180,E1 2689.178,E2 2689.178} C_VEL
LIN {X 0,Y 60.076,Z 1149.34,A -85,B 0,C 180,E1 2678.759,E2 2678.759} C_VEL
LIN {X 0,Y 44.099,Z 1152.063,A -85,B 0,C 180,E1 2662.524,E2 2662.524} C_VEL
LIN {X 0,Y 33.616,Z 1153.563,A -85,B 0,C 180,E1 2632.751,E2 2632.751} C_VEL
LIN {X 0,Y 32.155,Z 1153.811,A -85,B 0,C 180,E1 2610.004,E2 2610.004} C_VEL
LIN {X 0,Y 33.863,Z 1153.553,A -85,B 0,C 180,E1 2585.587,E2 2585.587} C_VEL
LIN {X 0,Y 44.735,Z 1151.99,A -85,B 0,C 180,E1 2556.43,E2 2556.43} C_VEL
LIN {X 0,Y 61.735,Z 1149.084,A -85,B 0,C 180,E1 2540.061,E2 2540.061} C_VEL
LIN {X 0,Y 82.347,Z 1144.317,A -85,B 0,C 180,E1 2530.427,E2 2530.427} C_VEL
LIN {X 0,Y 103.336,Z 1138.256,A -85,B 0,C 180,E1 2524.732,E2 2524.732} C_VEL
LIN {X 0,Y 123.645,Z 1130.863,A -85,B 0,C 180,E1 2521.058,E2 2521.058} C_VEL
LIN {X 0,Y 101.578,Z 1139.232,A -85,B 0,C 180,E1 2517.18,E2 2517.18} C_VEL
LIN {X 0,Y 80.51,Z 1145.673,A -85,B 0,C 180,E1 2511.431,E2 2511.431} C_VEL
LIN {X 0,Y 76.998,Z 1146.67,A -85,B 0,C 180,E1 2510.145,E2 2510.145} C_VEL
LIN {X 0,Y 69.922,Z 1148.464,A -85,B 0,C 180,E1 2508.075,E2 2508.075} C_VEL
LIN {X 0,Y 49.531,Z 1152.141,A -85,B 0,C 180,E1 2503.361,E2 2503.361} C_VEL
LIN {X 0,Y 43.676,Z 1152.997,A -85,B 0,C 180,E1 2499.545,E2 2499.545} C_VEL
LIN {X 0,Y 29.305,Z 1155.047,A -85,B 0,C 180,E1 2475.761,E2 2475.761} C_VEL
LIN {X 0,Y 24.108,Z 1155.827,A -85,B 0,C 180,E1 2439.544,E2 2439.544} C_VEL
LIN {X 0,Y 24.089,Z 1155.873,A -85,B 0,C 180,E1 2424.904,E2 2424.904} C_VEL
LIN {X 0,Y 28.04,Z 1155.216,A -85,B 0,C 180,E1 2388.481,E2 2388.481} C_VEL
LIN {X 0,Y 41.503,Z 1153.296,A -85,B 0,C 180,E1 2362.669,E2 2362.669} C_VEL
LIN {X 0,Y 62.656,Z 1149.415,A -85,B 0,C 180,E1 2348.338,E2 2348.338} C_VEL
LIN {X 0,Y 84.02,Z 1144.133,A -85,B 0,C 180,E1 2341.509,E2 2341.509} C_VEL
LIN {X 0,Y 97.247,Z 1140.176,A -85,B 0,C 180,E1 2338.78,E2 2338.78} C_VEL
LIN {X 0,Y 75.463,Z 1146.022,A -85,B 0,C 180,E1 2333.594,E2 2333.594} C_VEL
LIN {X 0,Y 53.993,Z 1150.249,A -85,B 0,C 180,E1 2324.364,E2 2324.364} C_VEL
LIN {X 0,Y 35.912,Z 1152.896,A -85,B 0,C 180,E1 2306.649,E2 2306.649} C_VEL
LIN {X 0,Y 25.413,Z 1153.918,A -85,B 0,C 180,E1 2273.174,E2 2273.174} C_VEL
LIN {X 0,Y 24.157,Z 1154.099,A -85,B 0,C 180,E1 2247.633,E2 2247.633} C_VEL
LIN {X 0,Y 27.543,Z 1153.781,A -85,B 0,C 180,E1 2214.497,E2 2214.497} C_VEL
LIN {X 0,Y 41.202,Z 1152.192,A -85,B 0,C 180,E1 2186.126,E2 2186.126} C_VEL
LIN {X 0,Y 61.261,Z 1149.072,A -85,B 0,C 180,E1 2171.691,E2 2171.691} C_VEL
LIN {X 0,Y 83.208,Z 1144.139,A -85,B 0,C 180,E1 2164.179,E2 2164.179} C_VEL
LIN {X 0,Y 97.004,Z 1140.327,A -85,B 0,C 180,E1 2161.152,E2 2161.152} C_VEL
LIN {X 0,Y 74.184,Z 1146.844,A -85,B 0,C 180,E1 2155.835,E2 2155.835} C_VEL
LIN {X 0,Y 52.474,Z 1151.459,A -85,B 0,C 180,E1 2146.345,E2 2146.345} C_VEL
LIN {X 0,Y 43.676,Z 1152.997,A -85,B 0,C 180,E1 2139.545,E2 2139.545} C_VEL
LIN {X 0,Y 37.081,Z 1153.918,A -85,B 0,C 180,E1 2133.85,E2 2133.85} C_VEL
LIN {X 0,Y 24.761,Z 1154.987,A -85,B 0,C 180,E1 2121.391,E2 2121.391} C_VEL
LIN {X 0,Y 17.425,Z 1155.411,A -85,B 0,C 180,E1 2099.913,E2 2099.913} C_VEL
LIN {X 0,Y 16.384,Z 1155.486,A -85,B 0,C 180,E1 2089.06,E2 2089.06} C_VEL
LIN {X 0,Y 16.097,Z 1155.601,A -85,B 0,C 180,E1 2066.431,E2 2066.431} C_VEL
LIN {X 0,Y 21.494,Z 1155.03,A -85,B 0,C 180,E1 2017.73,E2 2017.73} C_VEL
LIN {X 0,Y 38.043,Z 1153.121,A -85,B 0,C 180,E1 1992.134,E2 1992.134} C_VEL
LIN {X 0,Y 60.009,Z 1149.536,A -85,B 0,C 180,E1 1981.275,E2 1981.275} C_VEL
LIN {X 0,Y 69.604,Z 1147.445,A -85,B 0,C 180,E1 1978.664,E2 1978.664} C_VEL
LIN {X 0,Y 48.554,Z 1151.159,A -85,B 0,C 180,E1 1971.305,E2 1971.305} C_VEL
LIN {X 0,Y 28.003,Z 1153.518,A -85,B 0,C 180,E1 1953.215,E2 1953.215} C_VEL
LIN {X 0,Y 17.485,Z 1154.257,A -85,B 0,C 180,E1 1917.233,E2 1917.233} C_VEL
LIN {X 0,Y 16.216,Z 1154.378,A -85,B 0,C 180,E1 1882.924,E2 1882.924} C_VEL
LIN {X 0,Y 22.107,Z 1154.023,A -85,B 0,C 180,E1 1839.756,E2 1839.756} C_VEL
LIN {X 0,Y 38.306,Z 1152.499,A -85,B 0,C 180,E1 1815.045,E2 1815.045} C_VEL
LIN {X 0,Y 60.134,Z 1149.381,A -85,B 0,C 180,E1 1803.971,E2 1803.971} C_VEL
LIN {X 0,Y 69.451,Z 1147.527,A -85,B 0,C 180,E1 1801.295,E2 1801.295} C_VEL
LIN {X 0,Y 47.281,Z 1151.83,A -85,B 0,C 180,E1 1793.659,E2 1793.659} C_VEL
LIN {X 0,Y 26.604,Z 1154.507,A -85,B 0,C 180,E1 1774.41,E2 1774.41} C_VEL
LIN {X 0,Y 16.738,Z 1155.438,A -85,B 0,C 180,E1 1734.71,E2 1734.71} C_VEL
LIN {X 0,Y 16.384,Z 1155.486,A -85,B 0,C 180,E1 1729.06,E2 1729.06} C_VEL
LIN {X 0,Y 15.382,Z 1155.594,A -85,B 0,C 180,E1 1709.658,E2 1709.658} C_VEL
LIN {X 0,Y 14.814,Z 1155.391,A -85,B 0,C 180,E1 1682.163,E2 1682.163} C_VEL
LIN {X 0,Y 23.831,Z 1154.241,A -85,B 0,C 180,E1 1629.13,E2 1629.13} C_VEL
LIN {X 0,Y 27.984,Z 1153.878,A -85,B 0,C 180,E1 1624.578,E2 1624.578} C_VEL
LIN {X 0,Y 39.833,Z 1152.48,A -85,B 0,C 180,E1 1618.379,E2 1618.379} C_VEL
LIN {X 0,Y 20.733,Z 1154.127,A -85,B 0,C 180,E1 1604.714,E2 1604.714} C_VEL
LIN {X 0,Y 8.563,Z 1154.652,A -85,B 0,C 180,E1 1550.522,E2 1550.522} C_VEL
LIN {X 0,Y 9.29,Z 1154.62,A -85,B 0,C 180,E1 1497.46,E2 1497.46} C_VEL
LIN {X 0,Y 21.64,Z 1154.085,A -85,B 0,C 180,E1 1454.024,E2 1454.024} C_VEL
LIN {X 0,Y 39.848,Z 1152.509,A -85,B 0,C 180,E1 1441.531,E2 1441.531} C_VEL
LIN {X 0,Y 20.44,Z 1154.508,A -85,B 0,C 180,E1 1428.019,E2 1428.019} C_VEL
LIN {X 0,Y 8.158,Z 1155.278,A -85,B 0,C 180,E1 1364.174,E2 1364.174} C_VEL
LIN {X 0,Y 8.159,Z 1155.272,A -85,B 0,C 180,E1 1335.796,E2 1335.796} C_VEL
LIN {X 0,Y 20.444,Z 1154.491,A -85,B 0,C 180,E1 1271.969,E2 1271.969} C_VEL
LIN {X 0,Y 27.984,Z 1153.878,A -85,B 0,C 180,E1 1264.578,E2 1264.578} C_VEL
LIN {X 0,Y 26.948,Z 1153.915,A -85,B 0,C 180,E1 1262.465,E2 1262.465} C_VEL
LIN {X 0,Y 20.924,Z 1154.264,A -85,B 0,C 180,E1 1259.64,E2 1259.64} C_VEL
LIN {X 0,Y 5.588,Z 1154.903,A -85,B 0,C 180,E1 1256.116,E2 1256.116} C_VEL
LIN {X 0,Y 0.479,Z 1155.01,A -85,B 0,C 180,E1 1264.803,E2 1264.803} C_VEL
LIN {X 0,Y 1.374,Z 1154.993,A -85,B 0,C 180,E1 1443.227,E2 1443.227} C_VEL
LIN {X 0,Y 1.385,Z 1154.987,A -85,B 0,C 180,E1 1616.737,E2 1616.737} C_VEL
LIN {X 0,Y 0.479,Z 1155.01,A -85,B 0,C 180,E1 1624.803,E2 1624.803} C_VEL
LIN {X 0,Y 1.489,Z 1157.01,A -85,B 0,C 180,E1 1789.597,E2 1789.597} C_VEL
LIN {X 0,Y 1.489,Z 1180,A -85,B 0,C 180,E1 1789.597,E2 1789.597} C_VEL
LIN {X 0,Y 1.489,Z 1180,A -85,B 0,C 180,E1 1789.597,E2 1789.597}

QRS_NEXT_CUT()

QRS_NEXT()
QRS_HOME()

END
